LIN {X 0,Y 451.466,Z 366.784,A -85,B 0,C 180,E1 -8791.654,E2 -8791.654} C_VEL
LIN {X 0,Y 453.268,Z 375.362,A -85,B 0,C 180,E1 -8793.527,E2 -8793.527} C_VEL
LIN {X 0,Y 451.61,Z 393.058,A -85,B 0,C 180,E1 -8796.66,E2 -8796.66} C_VEL
LIN {X 0,Y 451.152,Z 398.451,A -85,B 0,C 180,E1 -8797.534,E2 -8797.534} C_VEL
LIN {X 0,Y 454.645,Z 414.595,A -85,B 0,C 180,E1 -8798.223,E2 -8798.223} C_VEL
LIN {X 0,Y 455.627,Z 420.756,A -85,B 0,C 180,E1 -8798.444,E2 -8798.444} C_VEL
LIN {X 0,Y 452.915,Z 505.565,A -85,B 0,C 180,E1 -8800.275,E2 -8800.275} C_VEL
LIN {X 0,Y 452.018,Z 542.086,A -85,B 0,C 180,E1 -8801.061,E2 -8801.061} C_VEL
LIN {X 0,Y 451.407,Z 557.431,A -85,B 0,C 180,E1 -8801.582,E2 -8801.582} C_VEL
LIN {X 0,Y 450.85,Z 571.274,A -85,B 0,C 180,E1 -8802.243,E2 -8802.243} C_VEL
LIN {X 0,Y 450.077,Z 585.059,A -85,B 0,C 180,E1 -8803.092,E2 -8803.092} C_VEL
LIN {X 0,Y 449.288,Z 598.112,A -85,B 0,C 180,E1 -8804.113,E2 -8804.113} C_VEL
LIN {X 0,Y 448.6,Z 609.92,A -85,B 0,C 180,E1 -8805.251,E2 -8805.251} C_VEL
LIN {X 0,Y 447.822,Z 620.998,A -85,B 0,C 180,E1 -8806.544,E2 -8806.544} C_VEL
LIN {X 0,Y 447.203,Z 631.086,A -85,B 0,C 180,E1 -8807.981,E2 -8807.981} C_VEL
LIN {X 0,Y 446.693,Z 638.983,A -85,B 0,C 180,E1 -8809.347,E2 -8809.347} C_VEL
LIN {X 0,Y 446.266,Z 646.534,A -85,B 0,C 180,E1 -8810.939,E2 -8810.939} C_VEL
LIN {X 0,Y 445.957,Z 651.754,A -85,B 0,C 180,E1 -8812.302,E2 -8812.302} C_VEL
LIN {X 0,Y 445.838,Z 655.972,A -85,B 0,C 180,E1 -8813.665,E2 -8813.665} C_VEL
LIN {X 0,Y 445.563,Z 660.212,A -85,B 0,C 180,E1 -8815.477,E2 -8815.477} C_VEL
LIN {X 0,Y 445.511,Z 662.951,A -85,B 0,C 180,E1 -8817.288,E2 -8817.288} C_VEL
LIN {X 0,Y 445.425,Z 664.278,A -85,B 0,C 180,E1 -8819.096,E2 -8819.096} C_VEL
LIN {X 0,Y 445.408,Z 664.199,A -85,B 0,C 180,E1 -8820.904,E2 -8820.904} C_VEL
LIN {X 0,Y 445.492,Z 662.715,A -85,B 0,C 180,E1 -8822.713,E2 -8822.713} C_VEL
LIN {X 0,Y 445.553,Z 661.444,A -85,B 0,C 180,E1 -8823.618,E2 -8823.618} C_VEL
LIN {X 0,Y 445.637,Z 657.807,A -85,B 0,C 180,E1 -8825.43,E2 -8825.43} C_VEL
LIN {X 0,Y 445.752,Z 654.529,A -85,B 0,C 180,E1 -8826.647,E2 -8826.647} C_VEL
LIN {X 0,Y 445.941,Z 649.406,A -85,B 0,C 180,E1 -8828.154,E2 -8828.154} C_VEL
LIN {X 0,Y 446.291,Z 642.628,A -85,B 0,C 180,E1 -8829.746,E2 -8829.746} C_VEL
LIN {X 0,Y 446.76,Z 634.19,A -85,B 0,C 180,E1 -8831.341,E2 -8831.341} C_VEL
LIN {X 0,Y 447.284,Z 625.36,A -85,B 0,C 180,E1 -8832.708,E2 -8832.708} C_VEL
LIN {X 0,Y 447.905,Z 614.653,A -85,B 0,C 180,E1 -8834.076,E2 -8834.076} C_VEL
LIN {X 0,Y 448.625,Z 602.694,A -85,B 0,C 180,E1 -8835.329,E2 -8835.329} C_VEL
LIN {X 0,Y 449.347,Z 590.755,A -85,B 0,C 180,E1 -8836.352,E2 -8836.352} C_VEL
LIN {X 0,Y 450.048,Z 577.658,A -85,B 0,C 180,E1 -8837.26,E2 -8837.26} C_VEL
LIN {X 0,Y 450.686,Z 563.753,A -85,B 0,C 180,E1 -8838.012,E2 -8838.012} C_VEL
LIN {X 0,Y 451.198,Z 549.271,A -85,B 0,C 180,E1 -8838.592,E2 -8838.592} C_VEL
LIN {X 0,Y 451.622,Z 534.731,A -85,B 0,C 180,E1 -8838.986,E2 -8838.986} C_VEL
LIN {X 0,Y 453.696,Z 419.17,A -85,B 0,C 180,E1 -8841.144,E2 -8841.144} C_VEL
LIN {X 0,Y 449.714,Z 397.572,A -85,B 0,C 180,E1 -8841.791,E2 -8841.791} C_VEL
LIN {X 0,Y 450.922,Z 378.264,A -85,B 0,C 180,E1 -8844.886,E2 -8844.886} C_VEL
LIN {X 0,Y 451.344,Z 370.862,A -85,B 0,C 180,E1 -8846.097,E2 -8846.097} C_VEL
LIN {X 0,Y 448.252,Z 357.222,A -85,B 0,C 180,E1 -8848.597,E2 -8848.597} C_VEL
LIN {X 0,Y 446.449,Z 349.788,A -85,B 0,C 180,E1 -8850.024,E2 -8850.024} C_VEL
LIN {X 0,Y 446.416,Z 349.503,A -85,B 0,C 180,E1 -8850.251,E2 -8850.251} C_VEL
LIN {X 0,Y 446.425,Z 349.502,A -85,B 0,C 180,E1 -8853.449,E2 -8853.449} C_VEL
LIN {X 0,Y 446.391,Z 349.505,A -85,B 0,C 180,E1 -8856.747,E2 -8856.747} C_VEL
LIN {X 0,Y 446.392,Z 349.508,A -85,B 0,C 180,E1 -8860.204,E2 -8860.204} C_VEL
LIN {X 0,Y 446.38,Z 349.497,A -85,B 0,C 180,E1 -8863.594,E2 -8863.594} C_VEL
LIN {X 0,Y 446.378,Z 349.497,A -85,B 0,C 180,E1 -8866.406,E2 -8866.406} C_VEL
LIN {X 0,Y 446.387,Z 349.503,A -85,B 0,C 180,E1 -8869.796,E2 -8869.796} C_VEL
LIN {X 0,Y 446.391,Z 349.499,A -85,B 0,C 180,E1 -8873.253,E2 -8873.253} C_VEL
LIN {X 0,Y 446.425,Z 349.504,A -85,B 0,C 180,E1 -8876.551,E2 -8876.551} C_VEL
LIN {X 0,Y 446.449,Z 349.719,A -85,B 0,C 180,E1 -8877.761,E2 -8877.761} C_VEL
LIN {X 0,Y 450.776,Z 366.42,A -85,B 0,C 180,E1 -8880.498,E2 -8880.498} C_VEL
LIN {X 0,Y 452.483,Z 374.302,A -85,B 0,C 180,E1 -8881.723,E2 -8881.723} C_VEL
LIN {X 0,Y 451.989,Z 384.049,A -85,B 0,C 180,E1 -8883.058,E2 -8883.058} C_VEL
LIN {X 0,Y 451.215,Z 387.102,A -85,B 0,C 180,E1 -8883.428,E2 -8883.428} C_VEL
LIN {X 0,Y 448.155,Z 392.329,A -85,B 0,C 180,E1 -8883.945,E2 -8883.945} C_VEL
LIN {X 0,Y 445.622,Z 397.396,A -85,B 0,C 180,E1 -8884.337,E2 -8884.337} C_VEL
LIN {X 0,Y 445.361,Z 400.297,A -85,B 0,C 180,E1 -8884.478,E2 -8884.478} C_VEL
LIN {X 0,Y 445.453,Z 400.893,A -85,B 0,C 180,E1 -8884.498,E2 -8884.498} C_VEL
LIN {X 0,Y 449.746,Z 423.038,A -85,B 0,C 180,E1 -8885.141,E2 -8885.141} C_VEL
LIN {X 0,Y 449.819,Z 431.74,A -85,B 0,C 180,E1 -8885.295,E2 -8885.295} C_VEL
LIN {X 0,Y 447.9,Z 564.075,A -85,B 0,C 180,E1 -8887.483,E2 -8887.483} C_VEL
LIN {X 0,Y 447.321,Z 579.57,A -85,B 0,C 180,E1 -8887.902,E2 -8887.902} C_VEL
LIN {X 0,Y 446.707,Z 592.8,A -85,B 0,C 180,E1 -8888.419,E2 -8888.419} C_VEL
LIN {X 0,Y 445.871,Z 606.369,A -85,B 0,C 180,E1 -8889.107,E2 -8889.107} C_VEL
LIN {X 0,Y 444.82,Z 620.534,A -85,B 0,C 180,E1 -8890.021,E2 -8890.021} C_VEL
LIN {X 0,Y 443.782,Z 633.454,A -85,B 0,C 180,E1 -8891.055,E2 -8891.055} C_VEL
LIN {X 0,Y 442.744,Z 645.813,A -85,B 0,C 180,E1 -8892.256,E2 -8892.256} C_VEL
LIN {X 0,Y 441.736,Z 657.318,A -85,B 0,C 180,E1 -8893.596,E2 -8893.596} C_VEL
LIN {X 0,Y 440.866,Z 667.346,A -85,B 0,C 180,E1 -8894.986,E2 -8894.986} C_VEL
LIN {X 0,Y 440.023,Z 677.147,A -85,B 0,C 180,E1 -8896.609,E2 -8896.609} C_VEL
LIN {X 0,Y 439.507,Z 685.285,A -85,B 0,C 180,E1 -8898.236,E2 -8898.236} C_VEL
LIN {X 0,Y 438.932,Z 692.025,A -85,B 0,C 180,E1 -8899.856,E2 -8899.856} C_VEL
LIN {X 0,Y 438.616,Z 698.269,A -85,B 0,C 180,E1 -8901.708,E2 -8901.708} C_VEL
LIN {X 0,Y 438.366,Z 703.48,A -85,B 0,C 180,E1 -8903.722,E2 -8903.722} C_VEL
LIN {X 0,Y 438.3,Z 706.652,A -85,B 0,C 180,E1 -8905.401,E2 -8905.401} C_VEL
LIN {X 0,Y 438.287,Z 708.995,A -85,B 0,C 180,E1 -8907.243,E2 -8907.243} C_VEL
LIN {X 0,Y 438.228,Z 710.186,A -85,B 0,C 180,E1 -8909.081,E2 -8909.081} C_VEL
LIN {X 0,Y 438.228,Z 710.202,A -85,B 0,C 180,E1 -8910.919,E2 -8910.919} C_VEL
LIN {X 0,Y 438.287,Z 709.07,A -85,B 0,C 180,E1 -8912.757,E2 -8912.757} C_VEL
LIN {X 0,Y 438.301,Z 706.79,A -85,B 0,C 180,E1 -8914.598,E2 -8914.598} C_VEL
LIN {X 0,Y 438.447,Z 703.314,A -85,B 0,C 180,E1 -8916.442,E2 -8916.442} C_VEL
LIN {X 0,Y 438.612,Z 698.552,A -85,B 0,C 180,E1 -8918.291,E2 -8918.291} C_VEL
LIN {X 0,Y 438.909,Z 692.375,A -85,B 0,C 180,E1 -8920.145,E2 -8920.145} C_VEL
LIN {X 0,Y 439.513,Z 684.613,A -85,B 0,C 180,E1 -8921.998,E2 -8921.998} C_VEL
LIN {X 0,Y 440.083,Z 676.342,A -85,B 0,C 180,E1 -8923.624,E2 -8923.624} C_VEL
LIN {X 0,Y 440.95,Z 666.376,A -85,B 0,C 180,E1 -8925.247,E2 -8925.247} C_VEL
LIN {X 0,Y 441.854,Z 656.204,A -85,B 0,C 180,E1 -8926.637,E2 -8926.637} C_VEL
LIN {X 0,Y 442.904,Z 644.034,A -85,B 0,C 180,E1 -8928.024,E2 -8928.024} C_VEL
LIN {X 0,Y 443.966,Z 631.862,A -85,B 0,C 180,E1 -8929.176,E2 -8929.176} C_VEL
LIN {X 0,Y 444.99,Z 618.593,A -85,B 0,C 180,E1 -8930.211,E2 -8930.211} C_VEL
LIN {X 0,Y 445.971,Z 604.954,A -85,B 0,C 180,E1 -8931.069,E2 -8931.069} C_VEL
LIN {X 0,Y 446.807,Z 589.736,A -85,B 0,C 180,E1 -8931.815,E2 -8931.815} C_VEL
LIN {X 0,Y 447.52,Z 575.51,A -85,B 0,C 180,E1 -8932.324,E2 -8932.324} C_VEL
LIN {X 0,Y 447.954,Z 560.083,A -85,B 0,C 180,E1 -8932.697,E2 -8932.697} C_VEL
LIN {X 0,Y 449.98,Z 425.271,A -85,B 0,C 180,E1 -8934.901,E2 -8934.901} C_VEL
LIN {X 0,Y 448.818,Z 417.732,A -85,B 0,C 180,E1 -8935.1,E2 -8935.1} C_VEL
LIN {X 0,Y 444.78,Z 397.136,A -85,B 0,C 180,E1 -8935.727,E2 -8935.727} C_VEL
LIN {X 0,Y 445.685,Z 378.356,A -85,B 0,C 180,E1 -8938.234,E2 -8938.234} C_VEL
LIN {X 0,Y 445.495,Z 374.677,A -85,B 0,C 180,E1 -8938.761,E2 -8938.761} C_VEL
LIN {X 0,Y 441.858,Z 359.718,A -85,B 0,C 180,E1 -8941.184,E2 -8941.184} C_VEL
LIN {X 0,Y 439.398,Z 350.524,A -85,B 0,C 180,E1 -8942.744,E2 -8942.744} C_VEL
LIN {X 0,Y 439.363,Z 350.373,A -85,B 0,C 180,E1 -8946.288,E2 -8946.288} C_VEL
LIN {X 0,Y 439.348,Z 350.379,A -85,B 0,C 180,E1 -8948.599,E2 -8948.599} C_VEL
LIN {X 0,Y 439.345,Z 350.381,A -85,B 0,C 180,E1 -8952.21,E2 -8952.21} C_VEL
LIN {X 0,Y 439.375,Z 350.376,A -85,B 0,C 180,E1 -8955.267,E2 -8955.267} C_VEL
LIN {X 0,Y 439.362,Z 350.38,A -85,B 0,C 180,E1 -8958.747,E2 -8958.747} C_VEL
LIN {X 0,Y 439.356,Z 350.379,A -85,B 0,C 180,E1 -8961.611,E2 -8961.611} C_VEL
LIN {X 0,Y 439.393,Z 350.369,A -85,B 0,C 180,E1 -8964.843,E2 -8964.843} C_VEL
LIN {X 0,Y 439.369,Z 350.372,A -85,B 0,C 180,E1 -8968.139,E2 -8968.139} C_VEL
LIN {X 0,Y 439.404,Z 350.374,A -85,B 0,C 180,E1 -8971.605,E2 -8971.605} C_VEL
LIN {X 0,Y 439.366,Z 350.378,A -85,B 0,C 180,E1 -8974.413,E2 -8974.413} C_VEL
LIN {X 0,Y 439.363,Z 350.373,A -85,B 0,C 180,E1 -8977.424,E2 -8977.424} C_VEL
LIN {X 0,Y 439.441,Z 350.368,A -85,B 0,C 180,E1 -8980.663,E2 -8980.663} C_VEL
LIN {X 0,Y 439.463,Z 350.363,A -85,B 0,C 180,E1 -8984.224,E2 -8984.224} C_VEL
LIN {X 0,Y 439.484,Z 350.356,A -85,B 0,C 180,E1 -8988.001,E2 -8988.001} C_VEL
LIN {X 0,Y 439.504,Z 350.365,A -85,B 0,C 180,E1 -8991.725,E2 -8991.725} C_VEL
LIN {X 0,Y 439.619,Z 350.337,A -85,B 0,C 180,E1 -8994.496,E2 -8994.496} C_VEL
LIN {X 0,Y 439.631,Z 350.345,A -85,B 0,C 180,E1 -8998.168,E2 -8998.168} C_VEL
LIN {X 0,Y 439.761,Z 350.323,A -85,B 0,C 180,E1 -9000,E2 -9000} C_VEL
LIN {X 0,Y 439.634,Z 350.337,A -85,B 0,C 180,E1 -9002.749,E2 -9002.749} C_VEL
LIN {X 0,Y 439.593,Z 350.344,A -85,B 0,C 180,E1 -9006.425,E2 -9006.425} C_VEL
LIN {X 0,Y 439.497,Z 350.356,A -85,B 0,C 180,E1 -9009.202,E2 -9009.202} C_VEL
LIN {X 0,Y 439.466,Z 350.361,A -85,B 0,C 180,E1 -9012.938,E2 -9012.938} C_VEL
LIN {X 0,Y 439.447,Z 350.367,A -85,B 0,C 180,E1 -9016.348,E2 -9016.348} C_VEL
LIN {X 0,Y 439.402,Z 350.365,A -85,B 0,C 180,E1 -9019.626,E2 -9019.626} C_VEL
LIN {X 0,Y 439.365,Z 350.379,A -85,B 0,C 180,E1 -9022.575,E2 -9022.575} C_VEL
LIN {X 0,Y 439.4,Z 350.371,A -85,B 0,C 180,E1 -9025.585,E2 -9025.585} C_VEL
LIN {X 0,Y 439.418,Z 350.374,A -85,B 0,C 180,E1 -9028.673,E2 -9028.673} C_VEL
LIN {X 0,Y 439.37,Z 350.378,A -85,B 0,C 180,E1 -9032.03,E2 -9032.03} C_VEL
LIN {X 0,Y 439.394,Z 350.376,A -85,B 0,C 180,E1 -9035.34,E2 -9035.34} C_VEL
LIN {X 0,Y 439.375,Z 350.366,A -85,B 0,C 180,E1 -9038.596,E2 -9038.596} C_VEL
LIN {X 0,Y 439.388,Z 350.355,A -85,B 0,C 180,E1 -9041.257,E2 -9041.257} C_VEL
LIN {X 0,Y 439.405,Z 350.373,A -85,B 0,C 180,E1 -9044.729,E2 -9044.729} C_VEL
LIN {X 0,Y 439.395,Z 350.364,A -85,B 0,C 180,E1 -9047.796,E2 -9047.796} C_VEL
LIN {X 0,Y 439.43,Z 350.372,A -85,B 0,C 180,E1 -9050.228,E2 -9050.228} C_VEL
LIN {X 0,Y 439.373,Z 350.378,A -85,B 0,C 180,E1 -9053.713,E2 -9053.713} C_VEL
LIN {X 0,Y 439.384,Z 350.38,A -85,B 0,C 180,E1 -9057.055,E2 -9057.055} C_VEL
LIN {X 0,Y 439.441,Z 350.626,A -85,B 0,C 180,E1 -9057.582,E2 -9057.582} C_VEL
LIN {X 0,Y 444.398,Z 368.974,A -85,B 0,C 180,E1 -9060.643,E2 -9060.643} C_VEL
LIN {X 0,Y 446.318,Z 376.633,A -85,B 0,C 180,E1 -9061.861,E2 -9061.861} C_VEL
LIN {X 0,Y 445.263,Z 391.914,A -85,B 0,C 180,E1 -9063.961,E2 -9063.961} C_VEL
LIN {X 0,Y 444.918,Z 396.826,A -85,B 0,C 180,E1 -9064.6,E2 -9064.6} C_VEL
LIN {X 0,Y 449.267,Z 422.728,A -85,B 0,C 180,E1 -9065.326,E2 -9065.326} C_VEL
LIN {X 0,Y 447.201,Z 564.707,A -85,B 0,C 180,E1 -9067.659,E2 -9067.659} C_VEL
LIN {X 0,Y 446.7,Z 580.228,A -85,B 0,C 180,E1 -9068.093,E2 -9068.093} C_VEL
LIN {X 0,Y 446.002,Z 594.377,A -85,B 0,C 180,E1 -9068.664,E2 -9068.664} C_VEL
LIN {X 0,Y 445.107,Z 608.773,A -85,B 0,C 180,E1 -9069.432,E2 -9069.432} C_VEL
LIN {X 0,Y 444.194,Z 622.326,A -85,B 0,C 180,E1 -9070.354,E2 -9070.354} C_VEL
LIN {X 0,Y 443.208,Z 634.778,A -85,B 0,C 180,E1 -9071.39,E2 -9071.39} C_VEL
LIN {X 0,Y 442.171,Z 647.145,A -85,B 0,C 180,E1 -9072.635,E2 -9072.635} C_VEL
LIN {X 0,Y 441.225,Z 658.798,A -85,B 0,C 180,E1 -9074.052,E2 -9074.052} C_VEL
LIN {X 0,Y 440.412,Z 668.389,A -85,B 0,C 180,E1 -9075.444,E2 -9075.444} C_VEL
LIN {X 0,Y 439.683,Z 677.782,A -85,B 0,C 180,E1 -9077.069,E2 -9077.069} C_VEL
LIN {X 0,Y 439.216,Z 685.58,A -85,B 0,C 180,E1 -9078.696,E2 -9078.696} C_VEL
LIN {X 0,Y 438.785,Z 692.041,A -85,B 0,C 180,E1 -9080.318,E2 -9080.318} C_VEL
LIN {X 0,Y 438.531,Z 697.96,A -85,B 0,C 180,E1 -9082.171,E2 -9082.171} C_VEL
LIN {X 0,Y 438.372,Z 701.809,A -85,B 0,C 180,E1 -9083.712,E2 -9083.712} C_VEL
LIN {X 0,Y 438.3,Z 704.995,A -85,B 0,C 180,E1 -9085.402,E2 -9085.402} C_VEL
LIN {X 0,Y 438.341,Z 707.327,A -85,B 0,C 180,E1 -9087.243,E2 -9087.243} C_VEL
LIN {X 0,Y 438.229,Z 708.501,A -85,B 0,C 180,E1 -9089.081,E2 -9089.081} C_VEL
LIN {X 0,Y 438.23,Z 708.501,A -85,B 0,C 180,E1 -9090.919,E2 -9090.919} C_VEL
LIN {X 0,Y 438.346,Z 707.329,A -85,B 0,C 180,E1 -9092.757,E2 -9092.757} C_VEL
LIN {X 0,Y 438.3,Z 704.996,A -85,B 0,C 180,E1 -9094.599,E2 -9094.599} C_VEL
LIN {X 0,Y 438.367,Z 701.445,A -85,B 0,C 180,E1 -9096.444,E2 -9096.444} C_VEL
LIN {X 0,Y 438.593,Z 696.593,A -85,B 0,C 180,E1 -9098.292,E2 -9098.292} C_VEL
LIN {X 0,Y 438.853,Z 690.314,A -85,B 0,C 180,E1 -9100.146,E2 -9100.146} C_VEL
LIN {X 0,Y 439.353,Z 683.524,A -85,B 0,C 180,E1 -9101.768,E2 -9101.768} C_VEL
LIN {X 0,Y 439.925,Z 675.307,A -85,B 0,C 180,E1 -9103.394,E2 -9103.394} C_VEL
LIN {X 0,Y 440.68,Z 665.392,A -85,B 0,C 180,E1 -9105.02,E2 -9105.02} C_VEL
LIN {X 0,Y 441.488,Z 655.224,A -85,B 0,C 180,E1 -9106.413,E2 -9106.413} C_VEL
LIN {X 0,Y 442.536,Z 643.3,A -85,B 0,C 180,E1 -9107.777,E2 -9107.777} C_VEL
LIN {X 0,Y 443.506,Z 630.878,A -85,B 0,C 180,E1 -9108.957,E2 -9108.957} C_VEL
LIN {X 0,Y 444.53,Z 617.563,A -85,B 0,C 180,E1 -9109.992,E2 -9109.992} C_VEL
LIN {X 0,Y 445.576,Z 602.772,A -85,B 0,C 180,E1 -9110.908,E2 -9110.908} C_VEL
LIN {X 0,Y 446.337,Z 588.561,A -85,B 0,C 180,E1 -9111.588,E2 -9111.588} C_VEL
LIN {X 0,Y 446.987,Z 573.017,A -85,B 0,C 180,E1 -9112.129,E2 -9112.129} C_VEL
LIN {X 0,Y 447.396,Z 556.928,A -85,B 0,C 180,E1 -9112.483,E2 -9112.483} C_VEL
LIN {X 0,Y 448.953,Z 450.43,A -85,B 0,C 180,E1 -9114.24,E2 -9114.24} C_VEL
LIN {X 0,Y 449.701,Z 421.272,A -85,B 0,C 180,E1 -9114.867,E2 -9114.867} C_VEL
LIN {X 0,Y 446.922,Z 403.458,A -85,B 0,C 180,E1 -9115.502,E2 -9115.502} C_VEL
LIN {X 0,Y 445.941,Z 398.268,A -85,B 0,C 180,E1 -9115.743,E2 -9115.743} C_VEL
LIN {X 0,Y 447.865,Z 381.434,A -85,B 0,C 180,E1 -9118.25,E2 -9118.25} C_VEL
LIN {X 0,Y 447.719,Z 378.874,A -85,B 0,C 180,E1 -9118.688,E2 -9118.688} C_VEL
LIN {X 0,Y 445.308,Z 368.642,A -85,B 0,C 180,E1 -9120.742,E2 -9120.742} C_VEL
LIN {X 0,Y 442.439,Z 359.291,A -85,B 0,C 180,E1 -9122.926,E2 -9122.926} C_VEL
LIN {X 0,Y 439.958,Z 352.426,A -85,B 0,C 180,E1 -9124.825,E2 -9124.825} C_VEL
LIN {X 0,Y 439.383,Z 350.43,A -85,B 0,C 180,E1 -9125.514,E2 -9125.514} C_VEL
LIN {X 0,Y 439.384,Z 350.381,A -85,B 0,C 180,E1 -9128.595,E2 -9128.595} C_VEL
LIN {X 0,Y 439.389,Z 350.38,A -85,B 0,C 180,E1 -9131.257,E2 -9131.257} C_VEL
LIN {X 0,Y 439.399,Z 350.379,A -85,B 0,C 180,E1 -9134.73,E2 -9134.73} C_VEL
LIN {X 0,Y 439.385,Z 350.38,A -85,B 0,C 180,E1 -9137.794,E2 -9137.794} C_VEL
LIN {X 0,Y 439.389,Z 350.38,A -85,B 0,C 180,E1 -9140.223,E2 -9140.223} C_VEL
LIN {X 0,Y 439.372,Z 350.382,A -85,B 0,C 180,E1 -9143.713,E2 -9143.713} C_VEL
LIN {X 0,Y 439.416,Z 350.546,A -85,B 0,C 180,E1 -9146.21,E2 -9146.21} C_VEL
LIN {X 0,Y 441.608,Z 357.326,A -85,B 0,C 180,E1 -9148.32,E2 -9148.32} C_VEL
LIN {X 0,Y 444.133,Z 365.947,A -85,B 0,C 180,E1 -9150.624,E2 -9150.624} C_VEL
LIN {X 0,Y 446.299,Z 375.378,A -85,B 0,C 180,E1 -9152.828,E2 -9152.828} C_VEL
LIN {X 0,Y 446.724,Z 377.823,A -85,B 0,C 180,E1 -9153.361,E2 -9153.361} C_VEL
LIN {X 0,Y 444.905,Z 395.726,A -85,B 0,C 180,E1 -9156.583,E2 -9156.583} C_VEL
LIN {X 0,Y 444.666,Z 398.418,A -85,B 0,C 180,E1 -9157.023,E2 -9157.023} C_VEL
LIN {X 0,Y 448.187,Z 414.555,A -85,B 0,C 180,E1 -9157.754,E2 -9157.754} C_VEL
LIN {X 0,Y 449.331,Z 422.382,A -85,B 0,C 180,E1 -9158.045,E2 -9158.045} C_VEL
LIN {X 0,Y 446.474,Z 504.686,A -85,B 0,C 180,E1 -9159.889,E2 -9159.889} C_VEL
LIN {X 0,Y 445.46,Z 542.04,A -85,B 0,C 180,E1 -9160.717,E2 -9160.717} C_VEL
LIN {X 0,Y 444.789,Z 557.63,A -85,B 0,C 180,E1 -9161.256,E2 -9161.256} C_VEL
LIN {X 0,Y 444.144,Z 572.359,A -85,B 0,C 180,E1 -9161.976,E2 -9161.976} C_VEL
LIN {X 0,Y 443.324,Z 585.762,A -85,B 0,C 180,E1 -9162.827,E2 -9162.827} C_VEL
LIN {X 0,Y 442.486,Z 598.72,A -85,B 0,C 180,E1 -9163.862,E2 -9163.862} C_VEL
LIN {X 0,Y 441.767,Z 610.473,A -85,B 0,C 180,E1 -9165.018,E2 -9165.018} C_VEL
LIN {X 0,Y 440.936,Z 621.682,A -85,B 0,C 180,E1 -9166.353,E2 -9166.353} C_VEL
LIN {X 0,Y 440.26,Z 631.568,A -85,B 0,C 180,E1 -9167.789,E2 -9167.789} C_VEL
LIN {X 0,Y 439.714,Z 639.451,A -85,B 0,C 180,E1 -9169.176,E2 -9169.176} C_VEL
LIN {X 0,Y 439.268,Z 646.975,A -85,B 0,C 180,E1 -9170.794,E2 -9170.794} C_VEL
LIN {X 0,Y 438.937,Z 652.19,A -85,B 0,C 180,E1 -9172.178,E2 -9172.178} C_VEL
LIN {X 0,Y 438.726,Z 657.628,A -85,B 0,C 180,E1 -9174.023,E2 -9174.023} C_VEL
LIN {X 0,Y 438.487,Z 660.621,A -85,B 0,C 180,E1 -9175.404,E2 -9175.404} C_VEL
LIN {X 0,Y 438.52,Z 662.157,A -85,B 0,C 180,E1 -9176.325,E2 -9176.325} C_VEL
LIN {X 0,Y 438.384,Z 664.168,A -85,B 0,C 180,E1 -9178.163,E2 -9178.163} C_VEL
LIN {X 0,Y 438.321,Z 664.766,A -85,B 0,C 180,E1 -9180,E2 -9180} C_VEL
LIN {X 0,Y 438.356,Z 663.945,A -85,B 0,C 180,E1 -9181.838,E2 -9181.838} C_VEL
LIN {X 0,Y 438.458,Z 661.718,A -85,B 0,C 180,E1 -9183.676,E2 -9183.676} C_VEL
LIN {X 0,Y 438.587,Z 658.035,A -85,B 0,C 180,E1 -9185.517,E2 -9185.517} C_VEL
LIN {X 0,Y 438.705,Z 654.282,A -85,B 0,C 180,E1 -9186.9,E2 -9186.9} C_VEL
LIN {X 0,Y 438.89,Z 649.55,A -85,B 0,C 180,E1 -9188.286,E2 -9188.286} C_VEL
LIN {X 0,Y 439.259,Z 642.708,A -85,B 0,C 180,E1 -9189.904,E2 -9189.904} C_VEL
LIN {X 0,Y 439.785,Z 634.172,A -85,B 0,C 180,E1 -9191.523,E2 -9191.523} C_VEL
LIN {X 0,Y 440.291,Z 625.257,A -85,B 0,C 180,E1 -9192.913,E2 -9192.913} C_VEL
LIN {X 0,Y 440.969,Z 614.452,A -85,B 0,C 180,E1 -9194.302,E2 -9194.302} C_VEL
LIN {X 0,Y 441.731,Z 602.379,A -85,B 0,C 180,E1 -9195.574,E2 -9195.574} C_VEL
LIN {X 0,Y 442.498,Z 590.311,A -85,B 0,C 180,E1 -9196.612,E2 -9196.612} C_VEL
LIN {X 0,Y 443.209,Z 577.038,A -85,B 0,C 180,E1 -9197.535,E2 -9197.535} C_VEL
LIN {X 0,Y 443.855,Z 563.864,A -85,B 0,C 180,E1 -9198.25,E2 -9198.25} C_VEL
LIN {X 0,Y 444.362,Z 549.683,A -85,B 0,C 180,E1 -9198.829,E2 -9198.829} C_VEL
LIN {X 0,Y 444.815,Z 535.354,A -85,B 0,C 180,E1 -9199.228,E2 -9199.228} C_VEL
LIN {X 0,Y 447.005,Z 420.277,A -85,B 0,C 180,E1 -9201.436,E2 -9201.436} C_VEL
LIN {X 0,Y 442.912,Z 397.889,A -85,B 0,C 180,E1 -9202.107,E2 -9202.107} C_VEL
LIN {X 0,Y 443.97,Z 381.108,A -85,B 0,C 180,E1 -9204.803,E2 -9204.803} C_VEL
LIN {X 0,Y 444.552,Z 373.397,A -85,B 0,C 180,E1 -9206.071,E2 -9206.071} C_VEL
LIN {X 0,Y 443.162,Z 366.192,A -85,B 0,C 180,E1 -9207.381,E2 -9207.381} C_VEL
LIN {X 0,Y 439.438,Z 350.774,A -85,B 0,C 180,E1 -9210.321,E2 -9210.321} C_VEL
LIN {X 0,Y 439.36,Z 350.41,A -85,B 0,C 180,E1 -9210.481,E2 -9210.481} C_VEL
LIN {X 0,Y 439.354,Z 350.385,A -85,B 0,C 180,E1 -9214.047,E2 -9214.047} C_VEL
LIN {X 0,Y 439.336,Z 350.384,A -85,B 0,C 180,E1 -9216.885,E2 -9216.885} C_VEL
LIN {X 0,Y 439.346,Z 350.385,A -85,B 0,C 180,E1 -9219.84,E2 -9219.84} C_VEL
LIN {X 0,Y 439.328,Z 350.371,A -85,B 0,C 180,E1 -9222.619,E2 -9222.619} C_VEL
LIN {X 0,Y 439.373,Z 350.379,A -85,B 0,C 180,E1 -9225.267,E2 -9225.267} C_VEL
LIN {X 0,Y 439.358,Z 350.382,A -85,B 0,C 180,E1 -9228.748,E2 -9228.748} C_VEL
LIN {X 0,Y 439.352,Z 350.381,A -85,B 0,C 180,E1 -9231.612,E2 -9231.612} C_VEL
LIN {X 0,Y 439.387,Z 350.378,A -85,B 0,C 180,E1 -9234.843,E2 -9234.843} C_VEL
LIN {X 0,Y 439.375,Z 350.524,A -85,B 0,C 180,E1 -9237.348,E2 -9237.348} C_VEL
LIN {X 0,Y 443.672,Z 366.741,A -85,B 0,C 180,E1 -9240.068,E2 -9240.068} C_VEL
LIN {X 0,Y 445.716,Z 375.854,A -85,B 0,C 180,E1 -9241.512,E2 -9241.512} C_VEL
LIN {X 0,Y 444.864,Z 394.937,A -85,B 0,C 180,E1 -9244.094,E2 -9244.094} C_VEL
LIN {X 0,Y 444.806,Z 397.613,A -85,B 0,C 180,E1 -9244.394,E2 -9244.394} C_VEL
LIN {X 0,Y 445.453,Z 400.893,A -85,B 0,C 180,E1 -9244.498,E2 -9244.498} C_VEL
LIN {X 0,Y 446.038,Z 406.682,A -85,B 0,C 180,E1 -9244.635,E2 -9244.635} C_VEL
LIN {X 0,Y 445.258,Z 416.52,A -85,B 0,C 180,E1 -9244.76,E2 -9244.76} C_VEL
LIN {X 0,Y 444.062,Z 424.472,A -85,B 0,C 180,E1 -9244.827,E2 -9244.827} C_VEL
LIN {X 0,Y 443.363,Z 432.441,A -85,B 0,C 180,E1 -9244.925,E2 -9244.925} C_VEL
LIN {X 0,Y 441.356,Z 563.988,A -85,B 0,C 180,E1 -9247.13,E2 -9247.13} C_VEL
LIN {X 0,Y 440.766,Z 578.845,A -85,B 0,C 180,E1 -9247.532,E2 -9247.532} C_VEL
LIN {X 0,Y 440.076,Z 592.717,A -85,B 0,C 180,E1 -9248.075,E2 -9248.075} C_VEL
LIN {X 0,Y 439.218,Z 606.337,A -85,B 0,C 180,E1 -9248.775,E2 -9248.775} C_VEL
LIN {X 0,Y 438.139,Z 620.508,A -85,B 0,C 180,E1 -9249.703,E2 -9249.703} C_VEL
LIN {X 0,Y 437.043,Z 633.431,A -85,B 0,C 180,E1 -9250.752,E2 -9250.752} C_VEL
LIN {X 0,Y 435.866,Z 646.524,A -85,B 0,C 180,E1 -9252.051,E2 -9252.051} C_VEL
LIN {X 0,Y 434.865,Z 657.3,A -85,B 0,C 180,E1 -9253.33,E2 -9253.33} C_VEL
LIN {X 0,Y 433.968,Z 667.329,A -85,B 0,C 180,E1 -9254.742,E2 -9254.742} C_VEL
LIN {X 0,Y 433.056,Z 677.131,A -85,B 0,C 180,E1 -9256.389,E2 -9256.389} C_VEL
LIN {X 0,Y 432.423,Z 686.315,A -85,B 0,C 180,E1 -9258.278,E2 -9258.278} C_VEL
LIN {X 0,Y 431.816,Z 693.728,A -85,B 0,C 180,E1 -9260.16,E2 -9260.16} C_VEL
LIN {X 0,Y 431.483,Z 699.612,A -85,B 0,C 180,E1 -9262.042,E2 -9262.042} C_VEL
LIN {X 0,Y 431.266,Z 703.781,A -85,B 0,C 180,E1 -9263.758,E2 -9263.758} C_VEL
LIN {X 0,Y 431.225,Z 706.638,A -85,B 0,C 180,E1 -9265.326,E2 -9265.326} C_VEL
LIN {X 0,Y 431.182,Z 708.981,A -85,B 0,C 180,E1 -9267.197,E2 -9267.197} C_VEL
LIN {X 0,Y 431.146,Z 710.173,A -85,B 0,C 180,E1 -9269.066,E2 -9269.066} C_VEL
LIN {X 0,Y 431.146,Z 710.188,A -85,B 0,C 180,E1 -9270.934,E2 -9270.934} C_VEL
LIN {X 0,Y 431.182,Z 709.055,A -85,B 0,C 180,E1 -9272.803,E2 -9272.803} C_VEL
LIN {X 0,Y 431.228,Z 706.776,A -85,B 0,C 180,E1 -9274.674,E2 -9274.674} C_VEL
LIN {X 0,Y 431.372,Z 703.299,A -85,B 0,C 180,E1 -9276.548,E2 -9276.548} C_VEL
LIN {X 0,Y 431.559,Z 698.535,A -85,B 0,C 180,E1 -9278.428,E2 -9278.428} C_VEL
LIN {X 0,Y 431.868,Z 692.357,A -85,B 0,C 180,E1 -9280.312,E2 -9280.312} C_VEL
LIN {X 0,Y 432.462,Z 685.691,A -85,B 0,C 180,E1 -9281.958,E2 -9281.958} C_VEL
LIN {X 0,Y 433.012,Z 677.615,A -85,B 0,C 180,E1 -9283.612,E2 -9283.612} C_VEL
LIN {X 0,Y 433.909,Z 667.916,A -85,B 0,C 180,E1 -9285.26,E2 -9285.26} C_VEL
LIN {X 0,Y 434.804,Z 657.98,A -85,B 0,C 180,E1 -9286.673,E2 -9286.673} C_VEL
LIN {X 0,Y 435.678,Z 648.071,A -85,B 0,C 180,E1 -9287.872,E2 -9287.872} C_VEL
LIN {X 0,Y 436.842,Z 635.672,A -85,B 0,C 180,E1 -9289.135,E2 -9289.135} C_VEL
LIN {X 0,Y 437.912,Z 623.225,A -85,B 0,C 180,E1 -9290.185,E2 -9290.185} C_VEL
LIN {X 0,Y 438.981,Z 609.727,A -85,B 0,C 180,E1 -9291.114,E2 -9291.114} C_VEL
LIN {X 0,Y 439.912,Z 595.638,A -85,B 0,C 180,E1 -9291.884,E2 -9291.884} C_VEL
LIN {X 0,Y 440.641,Z 581.153,A -85,B 0,C 180,E1 -9292.487,E2 -9292.487} C_VEL
LIN {X 0,Y 441.254,Z 566.778,A -85,B 0,C 180,E1 -9292.906,E2 -9292.906} C_VEL
LIN {X 0,Y 441.835,Z 533.359,A -85,B 0,C 180,E1 -9293.494,E2 -9293.494} C_VEL
LIN {X 0,Y 443.486,Z 424.86,A -85,B 0,C 180,E1 -9295.296,E2 -9295.296} C_VEL
LIN {X 0,Y 438.1,Z 397.116,A -85,B 0,C 180,E1 -9296.143,E2 -9296.143} C_VEL
LIN {X 0,Y 438.989,Z 379.693,A -85,B 0,C 180,E1 -9298.485,E2 -9298.485} C_VEL
LIN {X 0,Y 438.71,Z 376.309,A -85,B 0,C 180,E1 -9298.982,E2 -9298.982} C_VEL
LIN {X 0,Y 434.652,Z 359.737,A -85,B 0,C 180,E1 -9301.701,E2 -9301.701} C_VEL
LIN {X 0,Y 432.364,Z 351.363,A -85,B 0,C 180,E1 -9303.166,E2 -9303.166} C_VEL
LIN {X 0,Y 432.33,Z 351.249,A -85,B 0,C 180,E1 -9305.818,E2 -9305.818} C_VEL
LIN {X 0,Y 432.312,Z 351.253,A -85,B 0,C 180,E1 -9308.709,E2 -9308.709} C_VEL
LIN {X 0,Y 432.3,Z 351.263,A -85,B 0,C 180,E1 -9311.801,E2 -9311.801} C_VEL
LIN {X 0,Y 432.331,Z 351.255,A -85,B 0,C 180,E1 -9314.348,E2 -9314.348} C_VEL
LIN {X 0,Y 432.302,Z 351.261,A -85,B 0,C 180,E1 -9317.018,E2 -9317.018} C_VEL
LIN {X 0,Y 432.288,Z 351.264,A -85,B 0,C 180,E1 -9319.828,E2 -9319.828} C_VEL
LIN {X 0,Y 432.298,Z 351.26,A -85,B 0,C 180,E1 -9323.021,E2 -9323.021} C_VEL
LIN {X 0,Y 432.343,Z 351.257,A -85,B 0,C 180,E1 -9326,E2 -9326} C_VEL
LIN {X 0,Y 432.346,Z 351.25,A -85,B 0,C 180,E1 -9329.49,E2 -9329.49} C_VEL
LIN {X 0,Y 432.342,Z 351.249,A -85,B 0,C 180,E1 -9331.874,E2 -9331.874} C_VEL
LIN {X 0,Y 432.324,Z 351.255,A -85,B 0,C 180,E1 -9334.997,E2 -9334.997} C_VEL
LIN {X 0,Y 432.358,Z 351.244,A -85,B 0,C 180,E1 -9338.046,E2 -9338.046} C_VEL
LIN {X 0,Y 432.385,Z 351.249,A -85,B 0,C 180,E1 -9341.029,E2 -9341.029} C_VEL
LIN {X 0,Y 432.431,Z 351.237,A -85,B 0,C 180,E1 -9343.961,E2 -9343.961} C_VEL
LIN {X 0,Y 432.46,Z 351.232,A -85,B 0,C 180,E1 -9347.803,E2 -9347.803} C_VEL
LIN {X 0,Y 432.464,Z 351.243,A -85,B 0,C 180,E1 -9351.59,E2 -9351.59} C_VEL
LIN {X 0,Y 432.595,Z 351.212,A -85,B 0,C 180,E1 -9354.406,E2 -9354.406} C_VEL
LIN {X 0,Y 432.601,Z 351.221,A -85,B 0,C 180,E1 -9358.138,E2 -9358.138} C_VEL
LIN {X 0,Y 432.731,Z 351.199,A -85,B 0,C 180,E1 -9360,E2 -9360} C_VEL
LIN {X 0,Y 432.586,Z 351.215,A -85,B 0,C 180,E1 -9362.794,E2 -9362.794} C_VEL
LIN {X 0,Y 432.587,Z 351.222,A -85,B 0,C 180,E1 -9365.594,E2 -9365.594} C_VEL
LIN {X 0,Y 432.464,Z 351.226,A -85,B 0,C 180,E1 -9368.41,E2 -9368.41} C_VEL
LIN {X 0,Y 432.46,Z 351.233,A -85,B 0,C 180,E1 -9372.196,E2 -9372.196} C_VEL
LIN {X 0,Y 432.431,Z 351.241,A -85,B 0,C 180,E1 -9376.039,E2 -9376.039} C_VEL
LIN {X 0,Y 432.387,Z 351.238,A -85,B 0,C 180,E1 -9379.485,E2 -9379.485} C_VEL
LIN {X 0,Y 432.319,Z 351.261,A -85,B 0,C 180,E1 -9382.964,E2 -9382.964} C_VEL
LIN {X 0,Y 432.362,Z 351.247,A -85,B 0,C 180,E1 -9386.032,E2 -9386.032} C_VEL
LIN {X 0,Y 432.343,Z 351.249,A -85,B 0,C 180,E1 -9389.187,E2 -9389.187} C_VEL
LIN {X 0,Y 432.323,Z 351.257,A -85,B 0,C 180,E1 -9392.443,E2 -9392.443} C_VEL
LIN {X 0,Y 432.344,Z 351.255,A -85,B 0,C 180,E1 -9395.632,E2 -9395.632} C_VEL
LIN {X 0,Y 432.338,Z 351.239,A -85,B 0,C 180,E1 -9398.714,E2 -9398.714} C_VEL
LIN {X 0,Y 432.334,Z 351.243,A -85,B 0,C 180,E1 -9401.797,E2 -9401.797} C_VEL
LIN {X 0,Y 432.34,Z 351.255,A -85,B 0,C 180,E1 -9404.346,E2 -9404.346} C_VEL
LIN {X 0,Y 432.319,Z 351.236,A -85,B 0,C 180,E1 -9407.016,E2 -9407.016} C_VEL
LIN {X 0,Y 432.336,Z 351.255,A -85,B 0,C 180,E1 -9409.82,E2 -9409.82} C_VEL
LIN {X 0,Y 432.306,Z 351.262,A -85,B 0,C 180,E1 -9413.022,E2 -9413.022} C_VEL
LIN {X 0,Y 432.359,Z 351.256,A -85,B 0,C 180,E1 -9415.997,E2 -9415.997} C_VEL
LIN {X 0,Y 432.397,Z 351.504,A -85,B 0,C 180,E1 -9417.201,E2 -9417.201} C_VEL
LIN {X 0,Y 437.606,Z 370.765,A -85,B 0,C 180,E1 -9420.473,E2 -9420.473} C_VEL
LIN {X 0,Y 439.599,Z 379.254,A -85,B 0,C 180,E1 -9421.838,E2 -9421.838} C_VEL
LIN {X 0,Y 438.233,Z 396.054,A -85,B 0,C 180,E1 -9424.149,E2 -9424.149} C_VEL
LIN {X 0,Y 440.415,Z 408.746,A -85,B 0,C 180,E1 -9424.545,E2 -9424.545} C_VEL
LIN {X 0,Y 442.783,Z 424.102,A -85,B 0,C 180,E1 -9424.961,E2 -9424.961} C_VEL
LIN {X 0,Y 440.657,Z 564.835,A -85,B 0,C 180,E1 -9427.309,E2 -9427.309} C_VEL
LIN {X 0,Y 440.128,Z 580.292,A -85,B 0,C 180,E1 -9427.748,E2 -9427.748} C_VEL
LIN {X 0,Y 439.363,Z 594.732,A -85,B 0,C 180,E1 -9428.34,E2 -9428.34} C_VEL
LIN {X 0,Y 438.461,Z 608.817,A -85,B 0,C 180,E1 -9429.106,E2 -9429.106} C_VEL
LIN {X 0,Y 437.482,Z 622.362,A -85,B 0,C 180,E1 -9430.039,E2 -9430.039} C_VEL
LIN {X 0,Y 436.446,Z 634.808,A -85,B 0,C 180,E1 -9431.091,E2 -9431.091} C_VEL
LIN {X 0,Y 435.435,Z 646.391,A -85,B 0,C 180,E1 -9432.269,E2 -9432.269} C_VEL
LIN {X 0,Y 434.497,Z 657.047,A -85,B 0,C 180,E1 -9433.557,E2 -9433.557} C_VEL
LIN {X 0,Y 433.613,Z 666.931,A -85,B 0,C 180,E1 -9434.97,E2 -9434.97} C_VEL
LIN {X 0,Y 432.812,Z 676.575,A -85,B 0,C 180,E1 -9436.621,E2 -9436.621} C_VEL
LIN {X 0,Y 432.258,Z 684.593,A -85,B 0,C 180,E1 -9438.274,E2 -9438.274} C_VEL
LIN {X 0,Y 431.749,Z 692.058,A -85,B 0,C 180,E1 -9440.159,E2 -9440.159} C_VEL
LIN {X 0,Y 431.469,Z 697.976,A -85,B 0,C 180,E1 -9442.042,E2 -9442.042} C_VEL
LIN {X 0,Y 431.293,Z 702.081,A -85,B 0,C 180,E1 -9443.723,E2 -9443.723} C_VEL
LIN {X 0,Y 431.226,Z 705.009,A -85,B 0,C 180,E1 -9445.326,E2 -9445.326} C_VEL
LIN {X 0,Y 431.233,Z 707.341,A -85,B 0,C 180,E1 -9447.198,E2 -9447.198} C_VEL
LIN {X 0,Y 431.148,Z 708.514,A -85,B 0,C 180,E1 -9449.066,E2 -9449.066} C_VEL
LIN {X 0,Y 431.148,Z 708.515,A -85,B 0,C 180,E1 -9450.934,E2 -9450.934} C_VEL
LIN {X 0,Y 431.239,Z 707.343,A -85,B 0,C 180,E1 -9452.803,E2 -9452.803} C_VEL
LIN {X 0,Y 431.225,Z 705.01,A -85,B 0,C 180,E1 -9454.674,E2 -9454.674} C_VEL
LIN {X 0,Y 431.287,Z 701.459,A -85,B 0,C 180,E1 -9456.55,E2 -9456.55} C_VEL
LIN {X 0,Y 431.54,Z 696.608,A -85,B 0,C 180,E1 -9458.429,E2 -9458.429} C_VEL
LIN {X 0,Y 431.814,Z 690.329,A -85,B 0,C 180,E1 -9460.313,E2 -9460.313} C_VEL
LIN {X 0,Y 432.329,Z 683.54,A -85,B 0,C 180,E1 -9461.962,E2 -9461.962} C_VEL
LIN {X 0,Y 432.959,Z 675.323,A -85,B 0,C 180,E1 -9463.614,E2 -9463.614} C_VEL
LIN {X 0,Y 433.779,Z 665.411,A -85,B 0,C 180,E1 -9465.265,E2 -9465.265} C_VEL
LIN {X 0,Y 434.63,Z 655.244,A -85,B 0,C 180,E1 -9466.68,E2 -9466.68} C_VEL
LIN {X 0,Y 435.769,Z 643.102,A -85,B 0,C 180,E1 -9468.087,E2 -9468.087} C_VEL
LIN {X 0,Y 436.783,Z 630.903,A -85,B 0,C 180,E1 -9469.26,E2 -9469.26} C_VEL
LIN {X 0,Y 437.836,Z 617.593,A -85,B 0,C 180,E1 -9470.311,E2 -9470.311} C_VEL
LIN {X 0,Y 438.944,Z 602.809,A -85,B 0,C 180,E1 -9471.239,E2 -9471.239} C_VEL
LIN {X 0,Y 439.76,Z 588.31,A -85,B 0,C 180,E1 -9471.941,E2 -9471.941} C_VEL
LIN {X 0,Y 440.413,Z 573.165,A -85,B 0,C 180,E1 -9472.474,E2 -9472.474} C_VEL
LIN {X 0,Y 440.856,Z 557.05,A -85,B 0,C 180,E1 -9472.835,E2 -9472.835} C_VEL
LIN {X 0,Y 442.388,Z 459.964,A -85,B 0,C 180,E1 -9474.461,E2 -9474.461} C_VEL
LIN {X 0,Y 443.491,Z 422.194,A -85,B 0,C 180,E1 -9475.297,E2 -9475.297} C_VEL
LIN {X 0,Y 440.967,Z 405.481,A -85,B 0,C 180,E1 -9475.923,E2 -9475.923} C_VEL
LIN {X 0,Y 439.571,Z 398.326,A -85,B 0,C 180,E1 -9476.255,E2 -9476.255} C_VEL
LIN {X 0,Y 441.417,Z 383.429,A -85,B 0,C 180,E1 -9478.532,E2 -9478.532} C_VEL
LIN {X 0,Y 440.764,Z 379.01,A -85,B 0,C 180,E1 -9479.367,E2 -9479.367} C_VEL
LIN {X 0,Y 438.433,Z 369.61,A -85,B 0,C 180,E1 -9481.377,E2 -9481.377} C_VEL
LIN {X 0,Y 436.151,Z 362.168,A -85,B 0,C 180,E1 -9483.221,E2 -9483.221} C_VEL
LIN {X 0,Y 433.809,Z 355.65,A -85,B 0,C 180,E1 -9485.108,E2 -9485.108} C_VEL
LIN {X 0,Y 432.344,Z 351.339,A -85,B 0,C 180,E1 -9486.611,E2 -9486.611} C_VEL
LIN {X 0,Y 432.351,Z 351.257,A -85,B 0,C 180,E1 -9489.343,E2 -9489.343} C_VEL
LIN {X 0,Y 432.334,Z 351.258,A -85,B 0,C 180,E1 -9491.797,E2 -9491.797} C_VEL
LIN {X 0,Y 432.334,Z 351.259,A -85,B 0,C 180,E1 -9494.348,E2 -9494.348} C_VEL
LIN {X 0,Y 432.317,Z 351.261,A -85,B 0,C 180,E1 -9497.016,E2 -9497.016} C_VEL
LIN {X 0,Y 432.333,Z 351.259,A -85,B 0,C 180,E1 -9499.821,E2 -9499.821} C_VEL
LIN {X 0,Y 432.305,Z 351.263,A -85,B 0,C 180,E1 -9503.022,E2 -9503.022} C_VEL
LIN {X 0,Y 432.362,Z 351.414,A -85,B 0,C 180,E1 -9505.077,E2 -9505.077} C_VEL
LIN {X 0,Y 434.492,Z 357.608,A -85,B 0,C 180,E1 -9507.258,E2 -9507.258} C_VEL
LIN {X 0,Y 436.873,Z 365.418,A -85,B 0,C 180,E1 -9509.553,E2 -9509.553} C_VEL
LIN {X 0,Y 439.257,Z 375.188,A -85,B 0,C 180,E1 -9512.011,E2 -9512.011} C_VEL
LIN {X 0,Y 440.227,Z 380.402,A -85,B 0,C 180,E1 -9513.193,E2 -9513.193} C_VEL
LIN {X 0,Y 438.231,Z 398.139,A -85,B 0,C 180,E1 -9516.441,E2 -9516.441} C_VEL
LIN {X 0,Y 439.072,Z 402.188,A -85,B 0,C 180,E1 -9516.677,E2 -9516.677} C_VEL
LIN {X 0,Y 442.361,Z 417.597,A -85,B 0,C 180,E1 -9517.391,E2 -9517.391} C_VEL
LIN {X 0,Y 443.182,Z 422.812,A -85,B 0,C 180,E1 -9517.599,E2 -9517.599} C_VEL
LIN {X 0,Y 440.056,Z 504.347,A -85,B 0,C 180,E1 -9519.491,E2 -9519.491} C_VEL
LIN {X 0,Y 438.902,Z 543.015,A -85,B 0,C 180,E1 -9520.384,E2 -9520.384} C_VEL
LIN {X 0,Y 438.182,Z 558.408,A -85,B 0,C 180,E1 -9520.935,E2 -9520.935} C_VEL
LIN {X 0,Y 437.533,Z 572.066,A -85,B 0,C 180,E1 -9521.617,E2 -9521.617} C_VEL
LIN {X 0,Y 436.718,Z 585.008,A -85,B 0,C 180,E1 -9522.438,E2 -9522.438} C_VEL
LIN {X 0,Y 435.809,Z 598.141,A -85,B 0,C 180,E1 -9523.487,E2 -9523.487} C_VEL
LIN {X 0,Y 435.033,Z 610.031,A -85,B 0,C 180,E1 -9524.66,E2 -9524.66} C_VEL
LIN {X 0,Y 434.161,Z 620.844,A -85,B 0,C 180,E1 -9525.947,E2 -9525.947} C_VEL
LIN {X 0,Y 433.442,Z 630.611,A -85,B 0,C 180,E1 -9527.356,E2 -9527.356} C_VEL
LIN {X 0,Y 432.802,Z 638.716,A -85,B 0,C 180,E1 -9528.764,E2 -9528.764} C_VEL
LIN {X 0,Y 432.311,Z 646.463,A -85,B 0,C 180,E1 -9530.408,E2 -9530.408} C_VEL
LIN {X 0,Y 431.896,Z 652.66,A -85,B 0,C 180,E1 -9532.05,E2 -9532.05} C_VEL
LIN {X 0,Y 431.699,Z 656.844,A -85,B 0,C 180,E1 -9533.457,E2 -9533.457} C_VEL
LIN {X 0,Y 431.413,Z 661.045,A -85,B 0,C 180,E1 -9535.328,E2 -9535.328} C_VEL
LIN {X 0,Y 431.46,Z 662.569,A -85,B 0,C 180,E1 -9536.264,E2 -9536.264} C_VEL
LIN {X 0,Y 431.303,Z 664.557,A -85,B 0,C 180,E1 -9538.133,E2 -9538.133} C_VEL
LIN {X 0,Y 431.232,Z 665.116,A -85,B 0,C 180,E1 -9540,E2 -9540} C_VEL
LIN {X 0,Y 431.277,Z 664.254,A -85,B 0,C 180,E1 -9541.868,E2 -9541.868} C_VEL
LIN {X 0,Y 431.364,Z 661.984,A -85,B 0,C 180,E1 -9543.737,E2 -9543.737} C_VEL
LIN {X 0,Y 431.513,Z 658.25,A -85,B 0,C 180,E1 -9545.608,E2 -9545.608} C_VEL
LIN {X 0,Y 431.694,Z 652.957,A -85,B 0,C 180,E1 -9547.484,E2 -9547.484} C_VEL
LIN {X 0,Y 431.94,Z 647.829,A -85,B 0,C 180,E1 -9548.892,E2 -9548.892} C_VEL
LIN {X 0,Y 432.381,Z 640.454,A -85,B 0,C 180,E1 -9550.536,E2 -9550.536} C_VEL
LIN {X 0,Y 432.881,Z 632.73,A -85,B 0,C 180,E1 -9551.947,E2 -9551.947} C_VEL
LIN {X 0,Y 433.455,Z 623.269,A -85,B 0,C 180,E1 -9553.385,E2 -9553.385} C_VEL
LIN {X 0,Y 434.205,Z 612.214,A -85,B 0,C 180,E1 -9554.769,E2 -9554.769} C_VEL
LIN {X 0,Y 434.881,Z 600.809,A -85,B 0,C 180,E1 -9555.946,E2 -9555.946} C_VEL
LIN {X 0,Y 435.72,Z 588.265,A -85,B 0,C 180,E1 -9556.999,E2 -9556.999} C_VEL
LIN {X 0,Y 436.527,Z 574.516,A -85,B 0,C 180,E1 -9557.921,E2 -9557.921} C_VEL
LIN {X 0,Y 437.166,Z 559.956,A -85,B 0,C 180,E1 -9558.677,E2 -9558.677} C_VEL
LIN {X 0,Y 437.701,Z 545.674,A -85,B 0,C 180,E1 -9559.218,E2 -9559.218} C_VEL
LIN {X 0,Y 438.129,Z 530.368,A -85,B 0,C 180,E1 -9559.594,E2 -9559.594} C_VEL
LIN {X 0,Y 440.351,Z 421.289,A -85,B 0,C 180,E1 -9561.731,E2 -9561.731} C_VEL
LIN {X 0,Y 436.099,Z 397.76,A -85,B 0,C 180,E1 -9562.459,E2 -9562.459} C_VEL
LIN {X 0,Y 437.327,Z 379.438,A -85,B 0,C 180,E1 -9565.46,E2 -9565.46} C_VEL
LIN {X 0,Y 437.701,Z 374.813,A -85,B 0,C 180,E1 -9566.232,E2 -9566.232} C_VEL
LIN {X 0,Y 435.484,Z 364.439,A -85,B 0,C 180,E1 -9568.167,E2 -9568.167} C_VEL
LIN {X 0,Y 432.386,Z 351.714,A -85,B 0,C 180,E1 -9570.644,E2 -9570.644} C_VEL
LIN {X 0,Y 432.303,Z 351.266,A -85,B 0,C 180,E1 -9570.882,E2 -9570.882} C_VEL
LIN {X 0,Y 432.33,Z 351.26,A -85,B 0,C 180,E1 -9573.997,E2 -9573.997} C_VEL
LIN {X 0,Y 432.31,Z 351.259,A -85,B 0,C 180,E1 -9577.194,E2 -9577.194} C_VEL
LIN {X 0,Y 432.288,Z 351.265,A -85,B 0,C 180,E1 -9580.172,E2 -9580.172} C_VEL
LIN {X 0,Y 432.3,Z 351.247,A -85,B 0,C 180,E1 -9583.063,E2 -9583.063} C_VEL
LIN {X 0,Y 432.332,Z 351.257,A -85,B 0,C 180,E1 -9585.665,E2 -9585.665} C_VEL
LIN {X 0,Y 432.304,Z 351.263,A -85,B 0,C 180,E1 -9588.403,E2 -9588.403} C_VEL
LIN {X 0,Y 432.318,Z 351.26,A -85,B 0,C 180,E1 -9591.848,E2 -9591.848} C_VEL
LIN {X 0,Y 432.321,Z 351.255,A -85,B 0,C 180,E1 -9595.321,E2 -9595.321} C_VEL
LIN {X 0,Y 432.337,Z 351.476,A -85,B 0,C 180,E1 -9596.97,E2 -9596.97} C_VEL
LIN {X 0,Y 436.34,Z 366.42,A -85,B 0,C 180,E1 -9599.512,E2 -9599.512} C_VEL
LIN {X 0,Y 438.918,Z 377.432,A -85,B 0,C 180,E1 -9601.291,E2 -9601.291} C_VEL
LIN {X 0,Y 438.499,Z 388.448,A -85,B 0,C 180,E1 -9602.82,E2 -9602.82} C_VEL
LIN {X 0,Y 438.142,Z 397.417,A -85,B 0,C 180,E1 -9603.973,E2 -9603.973} C_VEL
LIN {X 0,Y 443.437,Z 424.846,A -85,B 0,C 180,E1 -9604.796,E2 -9604.796} C_VEL
LIN {X 0,Y 443.363,Z 432.441,A -85,B 0,C 180,E1 -9604.925,E2 -9604.925} C_VEL
LIN {X 0,Y 442.644,Z 438.297,A -85,B 0,C 180,E1 -9604.985,E2 -9604.985} C_VEL
LIN {X 0,Y 437.081,Z 457.362,A -85,B 0,C 180,E1 -9604.986,E2 -9604.986} C_VEL
LIN {X 0,Y 436.461,Z 463.211,A -85,B 0,C 180,E1 -9605.052,E2 -9605.052} C_VEL
LIN {X 0,Y 434.819,Z 563.902,A -85,B 0,C 180,E1 -9606.766,E2 -9606.766} C_VEL
LIN {X 0,Y 434.184,Z 579.373,A -85,B 0,C 180,E1 -9607.193,E2 -9607.193} C_VEL
LIN {X 0,Y 433.445,Z 593.531,A -85,B 0,C 180,E1 -9607.765,E2 -9607.765} C_VEL
LIN {X 0,Y 432.604,Z 606.305,A -85,B 0,C 180,E1 -9608.435,E2 -9608.435} C_VEL
LIN {X 0,Y 431.461,Z 620.481,A -85,B 0,C 180,E1 -9609.375,E2 -9609.375} C_VEL
LIN {X 0,Y 430.308,Z 633.408,A -85,B 0,C 180,E1 -9610.439,E2 -9610.439} C_VEL
LIN {X 0,Y 429.179,Z 645.56,A -85,B 0,C 180,E1 -9611.65,E2 -9611.65} C_VEL
LIN {X 0,Y 428.03,Z 657.282,A -85,B 0,C 180,E1 -9613.055,E2 -9613.055} C_VEL
LIN {X 0,Y 427.073,Z 667.312,A -85,B 0,C 180,E1 -9614.489,E2 -9614.489} C_VEL
LIN {X 0,Y 426.104,Z 677.115,A -85,B 0,C 180,E1 -9616.163,E2 -9616.163} C_VEL
LIN {X 0,Y 425.444,Z 685.255,A -85,B 0,C 180,E1 -9617.841,E2 -9617.841} C_VEL
LIN {X 0,Y 424.855,Z 691.996,A -85,B 0,C 180,E1 -9619.516,E2 -9619.516} C_VEL
LIN {X 0,Y 424.488,Z 698.241,A -85,B 0,C 180,E1 -9621.43,E2 -9621.43} C_VEL
LIN {X 0,Y 424.222,Z 703.076,A -85,B 0,C 180,E1 -9623.34,E2 -9623.34} C_VEL
LIN {X 0,Y 424.152,Z 706.625,A -85,B 0,C 180,E1 -9625.248,E2 -9625.248} C_VEL
LIN {X 0,Y 424.078,Z 708.968,A -85,B 0,C 180,E1 -9627.15,E2 -9627.15} C_VEL
LIN {X 0,Y 424.067,Z 710.159,A -85,B 0,C 180,E1 -9629.05,E2 -9629.05} C_VEL
LIN {X 0,Y 424.067,Z 710.174,A -85,B 0,C 180,E1 -9630.949,E2 -9630.949} C_VEL
LIN {X 0,Y 424.079,Z 709.041,A -85,B 0,C 180,E1 -9632.85,E2 -9632.85} C_VEL
LIN {X 0,Y 424.155,Z 706.761,A -85,B 0,C 180,E1 -9634.752,E2 -9634.752} C_VEL
LIN {X 0,Y 424.295,Z 703.283,A -85,B 0,C 180,E1 -9636.658,E2 -9636.658} C_VEL
LIN {X 0,Y 424.48,Z 698.518,A -85,B 0,C 180,E1 -9638.569,E2 -9638.569} C_VEL
LIN {X 0,Y 424.832,Z 692.339,A -85,B 0,C 180,E1 -9640.485,E2 -9640.485} C_VEL
LIN {X 0,Y 425.429,Z 685.672,A -85,B 0,C 180,E1 -9642.159,E2 -9642.159} C_VEL
LIN {X 0,Y 426.048,Z 677.595,A -85,B 0,C 180,E1 -9643.839,E2 -9643.839} C_VEL
LIN {X 0,Y 427.014,Z 667.893,A -85,B 0,C 180,E1 -9645.512,E2 -9645.512} C_VEL
LIN {X 0,Y 427.978,Z 657.955,A -85,B 0,C 180,E1 -9646.946,E2 -9646.946} C_VEL
LIN {X 0,Y 429.122,Z 646.159,A -85,B 0,C 180,E1 -9648.377,E2 -9648.377} C_VEL
LIN {X 0,Y 430.226,Z 634.377,A -85,B 0,C 180,E1 -9649.565,E2 -9649.565} C_VEL
LIN {X 0,Y 431.35,Z 621.647,A -85,B 0,C 180,E1 -9650.63,E2 -9650.63} C_VEL
LIN {X 0,Y 432.485,Z 607.763,A -85,B 0,C 180,E1 -9651.571,E2 -9651.571} C_VEL
LIN {X 0,Y 433.415,Z 593.738,A -85,B 0,C 180,E1 -9652.322,E2 -9652.322} C_VEL
LIN {X 0,Y 434.153,Z 579.668,A -85,B 0,C 180,E1 -9652.893,E2 -9652.893} C_VEL
LIN {X 0,Y 434.794,Z 563.942,A -85,B 0,C 180,E1 -9653.329,E2 -9653.329} C_VEL
LIN {X 0,Y 436.937,Z 435.773,A -85,B 0,C 180,E1 -9655.504,E2 -9655.504} C_VEL
LIN {X 0,Y 436.973,Z 425.414,A -85,B 0,C 180,E1 -9655.687,E2 -9655.687} C_VEL
LIN {X 0,Y 431.484,Z 397.43,A -85,B 0,C 180,E1 -9656.554,E2 -9656.554} C_VEL
LIN {X 0,Y 431.616,Z 392.802,A -85,B 0,C 180,E1 -9657.124,E2 -9657.124} C_VEL
LIN {X 0,Y 432.291,Z 380.675,A -85,B 0,C 180,E1 -9658.796,E2 -9658.796} C_VEL
LIN {X 0,Y 430.99,Z 373.972,A -85,B 0,C 180,E1 -9659.853,E2 -9659.853} C_VEL
LIN {X 0,Y 427.362,Z 359.675,A -85,B 0,C 180,E1 -9662.257,E2 -9662.257} C_VEL
LIN {X 0,Y 425.31,Z 352.269,A -85,B 0,C 180,E1 -9663.577,E2 -9663.577} C_VEL
LIN {X 0,Y 425.255,Z 352.131,A -85,B 0,C 180,E1 -9666.509,E2 -9666.509} C_VEL
LIN {X 0,Y 425.243,Z 352.129,A -85,B 0,C 180,E1 -9669.034,E2 -9669.034} C_VEL
LIN {X 0,Y 425.255,Z 352.135,A -85,B 0,C 180,E1 -9672.655,E2 -9672.655} C_VEL
LIN {X 0,Y 425.283,Z 352.131,A -85,B 0,C 180,E1 -9675.283,E2 -9675.283} C_VEL
LIN {X 0,Y 425.247,Z 352.139,A -85,B 0,C 180,E1 -9678.618,E2 -9678.618} C_VEL
LIN {X 0,Y 425.276,Z 352.13,A -85,B 0,C 180,E1 -9681.099,E2 -9681.099} C_VEL
LIN {X 0,Y 425.295,Z 352.125,A -85,B 0,C 180,E1 -9684.664,E2 -9684.664} C_VEL
LIN {X 0,Y 425.263,Z 352.129,A -85,B 0,C 180,E1 -9688.073,E2 -9688.073} C_VEL
LIN {X 0,Y 425.311,Z 352.133,A -85,B 0,C 180,E1 -9691.366,E2 -9691.366} C_VEL
LIN {X 0,Y 425.261,Z 352.135,A -85,B 0,C 180,E1 -9694.552,E2 -9694.552} C_VEL
LIN {X 0,Y 425.292,Z 352.124,A -85,B 0,C 180,E1 -9697.73,E2 -9697.73} C_VEL
LIN {X 0,Y 425.361,Z 352.122,A -85,B 0,C 180,E1 -9700.704,E2 -9700.704} C_VEL
LIN {X 0,Y 425.388,Z 352.111,A -85,B 0,C 180,E1 -9703.688,E2 -9703.688} C_VEL
LIN {X 0,Y 425.413,Z 352.112,A -85,B 0,C 180,E1 -9707.598,E2 -9707.598} C_VEL
LIN {X 0,Y 425.409,Z 352.119,A -85,B 0,C 180,E1 -9711.449,E2 -9711.449} C_VEL
LIN {X 0,Y 425.551,Z 352.089,A -85,B 0,C 180,E1 -9714.313,E2 -9714.313} C_VEL
LIN {X 0,Y 425.57,Z 352.097,A -85,B 0,C 180,E1 -9718.107,E2 -9718.107} C_VEL
LIN {X 0,Y 425.7,Z 352.074,A -85,B 0,C 180,E1 -9720,E2 -9720} C_VEL
LIN {X 0,Y 425.539,Z 352.093,A -85,B 0,C 180,E1 -9722.84,E2 -9722.84} C_VEL
LIN {X 0,Y 425.542,Z 352.098,A -85,B 0,C 180,E1 -9725.687,E2 -9725.687} C_VEL
LIN {X 0,Y 425.409,Z 352.104,A -85,B 0,C 180,E1 -9728.551,E2 -9728.551} C_VEL
LIN {X 0,Y 425.413,Z 352.111,A -85,B 0,C 180,E1 -9732.402,E2 -9732.402} C_VEL
LIN {X 0,Y 425.388,Z 352.118,A -85,B 0,C 180,E1 -9736.312,E2 -9736.312} C_VEL
LIN {X 0,Y 425.328,Z 352.117,A -85,B 0,C 180,E1 -9739.635,E2 -9739.635} C_VEL
LIN {X 0,Y 425.306,Z 352.129,A -85,B 0,C 180,E1 -9743.365,E2 -9743.365} C_VEL
LIN {X 0,Y 425.347,Z 352.125,A -85,B 0,C 180,E1 -9746.844,E2 -9746.844} C_VEL
LIN {X 0,Y 425.291,Z 352.123,A -85,B 0,C 180,E1 -9749.719,E2 -9749.719} C_VEL
LIN {X 0,Y 425.282,Z 352.135,A -85,B 0,C 180,E1 -9753.048,E2 -9753.048} C_VEL
LIN {X 0,Y 425.282,Z 352.133,A -85,B 0,C 180,E1 -9755.929,E2 -9755.929} C_VEL
LIN {X 0,Y 425.281,Z 352.11,A -85,B 0,C 180,E1 -9759.041,E2 -9759.041} C_VEL
LIN {X 0,Y 425.291,Z 352.123,A -85,B 0,C 180,E1 -9761.958,E2 -9761.958} C_VEL
LIN {X 0,Y 425.286,Z 352.122,A -85,B 0,C 180,E1 -9765.283,E2 -9765.283} C_VEL
LIN {X 0,Y 425.274,Z 352.13,A -85,B 0,C 180,E1 -9768.621,E2 -9768.621} C_VEL
LIN {X 0,Y 425.31,Z 352.135,A -85,B 0,C 180,E1 -9771.103,E2 -9771.103} C_VEL
LIN {X 0,Y 425.299,Z 352.135,A -85,B 0,C 180,E1 -9774.664,E2 -9774.664} C_VEL
LIN {X 0,Y 425.347,Z 352.363,A -85,B 0,C 180,E1 -9776.817,E2 -9776.817} C_VEL
LIN {X 0,Y 430.263,Z 370.521,A -85,B 0,C 180,E1 -9779.964,E2 -9779.964} C_VEL
LIN {X 0,Y 432.706,Z 380.443,A -85,B 0,C 180,E1 -9781.595,E2 -9781.595} C_VEL
LIN {X 0,Y 431.553,Z 395.549,A -85,B 0,C 180,E1 -9783.716,E2 -9783.716} C_VEL
LIN {X 0,Y 436.323,Z 423.881,A -85,B 0,C 180,E1 -9784.557,E2 -9784.557} C_VEL
LIN {X 0,Y 434.177,Z 563.487,A -85,B 0,C 180,E1 -9786.919,E2 -9786.919} C_VEL
LIN {X 0,Y 433.588,Z 578.523,A -85,B 0,C 180,E1 -9787.33,E2 -9787.33} C_VEL
LIN {X 0,Y 432.849,Z 592.282,A -85,B 0,C 180,E1 -9787.875,E2 -9787.875} C_VEL
LIN {X 0,Y 431.993,Z 606.888,A -85,B 0,C 180,E1 -9788.653,E2 -9788.653} C_VEL
LIN {X 0,Y 430.861,Z 620.824,A -85,B 0,C 180,E1 -9789.595,E2 -9789.595} C_VEL
LIN {X 0,Y 429.825,Z 633.553,A -85,B 0,C 180,E1 -9790.664,E2 -9790.664} C_VEL
LIN {X 0,Y 428.743,Z 645.307,A -85,B 0,C 180,E1 -9791.853,E2 -9791.853} C_VEL
LIN {X 0,Y 427.649,Z 657.071,A -85,B 0,C 180,E1 -9793.286,E2 -9793.286} C_VEL
LIN {X 0,Y 426.7,Z 666.952,A -85,B 0,C 180,E1 -9794.721,E2 -9794.721} C_VEL
LIN {X 0,Y 425.858,Z 676.595,A -85,B 0,C 180,E1 -9796.398,E2 -9796.398} C_VEL
LIN {X 0,Y 425.252,Z 684.612,A -85,B 0,C 180,E1 -9798.078,E2 -9798.078} C_VEL
LIN {X 0,Y 424.693,Z 692.075,A -85,B 0,C 180,E1 -9799.994,E2 -9799.994} C_VEL
LIN {X 0,Y 424.4,Z 697.992,A -85,B 0,C 180,E1 -9801.908,E2 -9801.908} C_VEL
LIN {X 0,Y 424.194,Z 702.403,A -85,B 0,C 180,E1 -9803.759,E2 -9803.759} C_VEL
LIN {X 0,Y 424.153,Z 705.024,A -85,B 0,C 180,E1 -9805.248,E2 -9805.248} C_VEL
LIN {X 0,Y 424.127,Z 707.355,A -85,B 0,C 180,E1 -9807.151,E2 -9807.151} C_VEL
LIN {X 0,Y 424.069,Z 708.528,A -85,B 0,C 180,E1 -9809.051,E2 -9809.051} C_VEL
LIN {X 0,Y 424.069,Z 708.528,A -85,B 0,C 180,E1 -9810.95,E2 -9810.95} C_VEL
LIN {X 0,Y 424.132,Z 707.357,A -85,B 0,C 180,E1 -9812.85,E2 -9812.85} C_VEL
LIN {X 0,Y 424.152,Z 705.023,A -85,B 0,C 180,E1 -9814.752,E2 -9814.752} C_VEL
LIN {X 0,Y 424.22,Z 701.473,A -85,B 0,C 180,E1 -9816.66,E2 -9816.66} C_VEL
LIN {X 0,Y 424.46,Z 696.622,A -85,B 0,C 180,E1 -9818.57,E2 -9818.57} C_VEL
LIN {X 0,Y 424.781,Z 690.344,A -85,B 0,C 180,E1 -9820.486,E2 -9820.486} C_VEL
LIN {X 0,Y 425.311,Z 683.556,A -85,B 0,C 180,E1 -9822.163,E2 -9822.163} C_VEL
LIN {X 0,Y 425.979,Z 675.34,A -85,B 0,C 180,E1 -9823.841,E2 -9823.841} C_VEL
LIN {X 0,Y 426.858,Z 665.429,A -85,B 0,C 180,E1 -9825.519,E2 -9825.519} C_VEL
LIN {X 0,Y 427.8,Z 655.263,A -85,B 0,C 180,E1 -9826.954,E2 -9826.954} C_VEL
LIN {X 0,Y 428.986,Z 643.124,A -85,B 0,C 180,E1 -9828.383,E2 -9828.383} C_VEL
LIN {X 0,Y 430.053,Z 630.928,A -85,B 0,C 180,E1 -9829.574,E2 -9829.574} C_VEL
LIN {X 0,Y 431.173,Z 617.622,A -85,B 0,C 180,E1 -9830.639,E2 -9830.639} C_VEL
LIN {X 0,Y 432.288,Z 602.845,A -85,B 0,C 180,E1 -9831.582,E2 -9831.582} C_VEL
LIN {X 0,Y 433.195,Z 587.723,A -85,B 0,C 180,E1 -9832.319,E2 -9832.319} C_VEL
LIN {X 0,Y 433.868,Z 572.594,A -85,B 0,C 180,E1 -9832.851,E2 -9832.851} C_VEL
LIN {X 0,Y 434.323,Z 557.169,A -85,B 0,C 180,E1 -9833.199,E2 -9833.199} C_VEL
LIN {X 0,Y 435.724,Z 470.922,A -85,B 0,C 180,E1 -9834.668,E2 -9834.668} C_VEL
LIN {X 0,Y 437.366,Z 423.399,A -85,B 0,C 180,E1 -9835.742,E2 -9835.742} C_VEL
LIN {X 0,Y 434.955,Z 407.01,A -85,B 0,C 180,E1 -9836.383,E2 -9836.383} C_VEL
LIN {X 0,Y 433.248,Z 398.473,A -85,B 0,C 180,E1 -9836.787,E2 -9836.787} C_VEL
LIN {X 0,Y 434.926,Z 386.063,A -85,B 0,C 180,E1 -9838.733,E2 -9838.733} C_VEL
LIN {X 0,Y 434.764,Z 383.519,A -85,B 0,C 180,E1 -9839.201,E2 -9839.201} C_VEL
LIN {X 0,Y 432.451,Z 373.67,A -85,B 0,C 180,E1 -9841.336,E2 -9841.336} C_VEL
LIN {X 0,Y 429.893,Z 365.11,A -85,B 0,C 180,E1 -9843.513,E2 -9843.513} C_VEL
LIN {X 0,Y 427.512,Z 358.419,A -85,B 0,C 180,E1 -9845.569,E2 -9845.569} C_VEL
LIN {X 0,Y 425.326,Z 352.277,A -85,B 0,C 180,E1 -9847.914,E2 -9847.914} C_VEL
LIN {X 0,Y 425.275,Z 352.138,A -85,B 0,C 180,E1 -9851.379,E2 -9851.379} C_VEL
LIN {X 0,Y 425.285,Z 352.137,A -85,B 0,C 180,E1 -9854.717,E2 -9854.717} C_VEL
LIN {X 0,Y 425.283,Z 352.137,A -85,B 0,C 180,E1 -9858.043,E2 -9858.043} C_VEL
LIN {X 0,Y 425.292,Z 352.136,A -85,B 0,C 180,E1 -9861.101,E2 -9861.101} C_VEL
LIN {X 0,Y 425.295,Z 352.364,A -85,B 0,C 180,E1 -9863.742,E2 -9863.742} C_VEL
LIN {X 0,Y 427.317,Z 357.846,A -85,B 0,C 180,E1 -9866,E2 -9866} C_VEL
LIN {X 0,Y 429.667,Z 365.273,A -85,B 0,C 180,E1 -9868.438,E2 -9868.438} C_VEL
LIN {X 0,Y 431.601,Z 372.486,A -85,B 0,C 180,E1 -9870.457,E2 -9870.457} C_VEL
LIN {X 0,Y 433.604,Z 381.799,A -85,B 0,C 180,E1 -9872.749,E2 -9872.749} C_VEL
LIN {X 0,Y 433.571,Z 384.418,A -85,B 0,C 180,E1 -9873.294,E2 -9873.294} C_VEL
LIN {X 0,Y 431.876,Z 398.63,A -85,B 0,C 180,E1 -9875.915,E2 -9875.915} C_VEL
LIN {X 0,Y 435.461,Z 414.542,A -85,B 0,C 180,E1 -9876.738,E2 -9876.738} C_VEL
LIN {X 0,Y 437.036,Z 424.563,A -85,B 0,C 180,E1 -9877.16,E2 -9877.16} C_VEL
LIN {X 0,Y 433.646,Z 505.765,A -85,B 0,C 180,E1 -9879.112,E2 -9879.112} C_VEL
LIN {X 0,Y 432.413,Z 543.352,A -85,B 0,C 180,E1 -9880.012,E2 -9880.012} C_VEL
LIN {X 0,Y 431.649,Z 558.18,A -85,B 0,C 180,E1 -9880.551,E2 -9880.551} C_VEL
LIN {X 0,Y 430.899,Z 573.262,A -85,B 0,C 180,E1 -9881.322,E2 -9881.322} C_VEL
LIN {X 0,Y 429.883,Z 587.524,A -85,B 0,C 180,E1 -9882.272,E2 -9882.272} C_VEL
LIN {X 0,Y 428.942,Z 600.227,A -85,B 0,C 180,E1 -9883.338,E2 -9883.338} C_VEL
LIN {X 0,Y 428.13,Z 611.818,A -85,B 0,C 180,E1 -9884.529,E2 -9884.529} C_VEL
LIN {X 0,Y 427.172,Z 623.17,A -85,B 0,C 180,E1 -9885.941,E2 -9885.941} C_VEL
LIN {X 0,Y 426.406,Z 632.687,A -85,B 0,C 180,E1 -9887.386,E2 -9887.386} C_VEL
LIN {X 0,Y 425.784,Z 640.508,A -85,B 0,C 180,E1 -9888.817,E2 -9888.817} C_VEL
LIN {X 0,Y 425.287,Z 647.955,A -85,B 0,C 180,E1 -9890.488,E2 -9890.488} C_VEL
LIN {X 0,Y 424.871,Z 653.157,A -85,B 0,C 180,E1 -9891.917,E2 -9891.917} C_VEL
LIN {X 0,Y 424.649,Z 657.312,A -85,B 0,C 180,E1 -9893.347,E2 -9893.347} C_VEL
LIN {X 0,Y 424.342,Z 661.486,A -85,B 0,C 180,E1 -9895.25,E2 -9895.25} C_VEL
LIN {X 0,Y 424.401,Z 662.997,A -85,B 0,C 180,E1 -9896.202,E2 -9896.202} C_VEL
LIN {X 0,Y 424.226,Z 664.95,A -85,B 0,C 180,E1 -9898.101,E2 -9898.101} C_VEL
LIN {X 0,Y 424.145,Z 665.463,A -85,B 0,C 180,E1 -9900,E2 -9900} C_VEL
LIN {X 0,Y 424.201,Z 664.559,A -85,B 0,C 180,E1 -9901.899,E2 -9901.899} C_VEL
LIN {X 0,Y 424.283,Z 663.578,A -85,B 0,C 180,E1 -9902.848,E2 -9902.848} C_VEL
LIN {X 0,Y 424.3,Z 660.537,A -85,B 0,C 180,E1 -9904.751,E2 -9904.751} C_VEL
LIN {X 0,Y 424.508,Z 656.873,A -85,B 0,C 180,E1 -9906.329,E2 -9906.329} C_VEL
LIN {X 0,Y 424.7,Z 651.471,A -85,B 0,C 180,E1 -9908.086,E2 -9908.086} C_VEL
LIN {X 0,Y 425.096,Z 644.903,A -85,B 0,C 180,E1 -9909.757,E2 -9909.757} C_VEL
LIN {X 0,Y 425.584,Z 636.719,A -85,B 0,C 180,E1 -9911.43,E2 -9911.43} C_VEL
LIN {X 0,Y 426.204,Z 628.168,A -85,B 0,C 180,E1 -9912.863,E2 -9912.863} C_VEL
LIN {X 0,Y 426.844,Z 617.866,A -85,B 0,C 180,E1 -9914.299,E2 -9914.299} C_VEL
LIN {X 0,Y 427.616,Z 606.402,A -85,B 0,C 180,E1 -9915.612,E2 -9915.612} C_VEL
LIN {X 0,Y 428.493,Z 593.593,A -85,B 0,C 180,E1 -9916.803,E2 -9916.803} C_VEL
LIN {X 0,Y 429.272,Z 580.971,A -85,B 0,C 180,E1 -9917.754,E2 -9917.754} C_VEL
LIN {X 0,Y 430.063,Z 566.568,A -85,B 0,C 180,E1 -9918.609,E2 -9918.609} C_VEL
LIN {X 0,Y 430.665,Z 551.846,A -85,B 0,C 180,E1 -9919.266,E2 -9919.266} C_VEL
LIN {X 0,Y 431.155,Z 537.375,A -85,B 0,C 180,E1 -9919.707,E2 -9919.707} C_VEL
LIN {X 0,Y 433.733,Z 422.943,A -85,B 0,C 180,E1 -9922.014,E2 -9922.014} C_VEL
LIN {X 0,Y 429.263,Z 397.866,A -85,B 0,C 180,E1 -9922.793,E2 -9922.793} C_VEL
LIN {X 0,Y 430.492,Z 380.729,A -85,B 0,C 180,E1 -9925.634,E2 -9925.634} C_VEL
LIN {X 0,Y 430.859,Z 376.416,A -85,B 0,C 180,E1 -9926.365,E2 -9926.365} C_VEL
LIN {X 0,Y 428.515,Z 365.683,A -85,B 0,C 180,E1 -9928.4,E2 -9928.4} C_VEL
LIN {X 0,Y 425.302,Z 352.46,A -85,B 0,C 180,E1 -9931.022,E2 -9931.022} C_VEL
LIN {X 0,Y 425.261,Z 352.141,A -85,B 0,C 180,E1 -9931.371,E2 -9931.371} C_VEL
LIN {X 0,Y 425.288,Z 352.137,A -85,B 0,C 180,E1 -9934.283,E2 -9934.283} C_VEL
LIN {X 0,Y 425.269,Z 352.138,A -85,B 0,C 180,E1 -9937.695,E2 -9937.695} C_VEL
LIN {X 0,Y 425.241,Z 352.139,A -85,B 0,C 180,E1 -9940.514,E2 -9940.514} C_VEL
LIN {X 0,Y 425.244,Z 352.128,A -85,B 0,C 180,E1 -9943.349,E2 -9943.349} C_VEL
LIN {X 0,Y 425.255,Z 352.131,A -85,B 0,C 180,E1 -9946.043,E2 -9946.043} C_VEL
LIN {X 0,Y 425.245,Z 352.141,A -85,B 0,C 180,E1 -9948.618,E2 -9948.618} C_VEL
LIN {X 0,Y 425.269,Z 352.136,A -85,B 0,C 180,E1 -9952.304,E2 -9952.304} C_VEL
LIN {X 0,Y 425.282,Z 352.131,A -85,B 0,C 180,E1 -9955.815,E2 -9955.815} C_VEL
LIN {X 0,Y 425.321,Z 352.397,A -85,B 0,C 180,E1 -9956.566,E2 -9956.566} C_VEL
LIN {X 0,Y 429.583,Z 368.282,A -85,B 0,C 180,E1 -9959.299,E2 -9959.299} C_VEL
LIN {X 0,Y 432.276,Z 379.918,A -85,B 0,C 180,E1 -9961.199,E2 -9961.199} C_VEL
LIN {X 0,Y 431.498,Z 397.119,A -85,B 0,C 180,E1 -9963.53,E2 -9963.53} C_VEL
LIN {X 0,Y 436.987,Z 425.671,A -85,B 0,C 180,E1 -9964.414,E2 -9964.414} C_VEL
LIN {X 0,Y 436.461,Z 463.211,A -85,B 0,C 180,E1 -9965.052,E2 -9965.052} C_VEL
LIN {X 0,Y 435.846,Z 469.057,A -85,B 0,C 180,E1 -9965.119,E2 -9965.119} C_VEL
LIN {X 0,Y 430.288,Z 488.115,A -85,B 0,C 180,E1 -9965.122,E2 -9965.122} C_VEL
LIN {X 0,Y 429.547,Z 493.97,A -85,B 0,C 180,E1 -9965.182,E2 -9965.182} C_VEL
LIN {X 0,Y 428.258,Z 565.172,A -85,B 0,C 180,E1 -9966.421,E2 -9966.421} C_VEL
LIN {X 0,Y 427.594,Z 580.526,A -85,B 0,C 180,E1 -9966.867,E2 -9966.867} C_VEL
LIN {X 0,Y 426.814,Z 594.299,A -85,B 0,C 180,E1 -9967.442,E2 -9967.442} C_VEL
LIN {X 0,Y 425.85,Z 608.195,A -85,B 0,C 180,E1 -9968.202,E2 -9968.202} C_VEL
LIN {X 0,Y 424.671,Z 621.994,A -85,B 0,C 180,E1 -9969.157,E2 -9969.157} C_VEL
LIN {X 0,Y 423.337,Z 635.909,A -85,B 0,C 180,E1 -9970.356,E2 -9970.356} C_VEL
LIN {X 0,Y 422.116,Z 647.994,A -85,B 0,C 180,E1 -9971.626,E2 -9971.626} C_VEL
LIN {X 0,Y 420.991,Z 659.015,A -85,B 0,C 180,E1 -9973.013,E2 -9973.013} C_VEL
LIN {X 0,Y 420.019,Z 668.776,A -85,B 0,C 180,E1 -9974.471,E2 -9974.471} C_VEL
LIN {X 0,Y 419.035,Z 678.326,A -85,B 0,C 180,E1 -9976.172,E2 -9976.172} C_VEL
LIN {X 0,Y 418.389,Z 686.286,A -85,B 0,C 180,E1 -9977.879,E2 -9977.879} C_VEL
LIN {X 0,Y 417.718,Z 693.699,A -85,B 0,C 180,E1 -9979.825,E2 -9979.825} C_VEL
LIN {X 0,Y 417.361,Z 699.585,A -85,B 0,C 180,E1 -9981.771,E2 -9981.771} C_VEL
LIN {X 0,Y 417.105,Z 704.238,A -85,B 0,C 180,E1 -9983.784,E2 -9983.784} C_VEL
LIN {X 0,Y 417.058,Z 706.611,A -85,B 0,C 180,E1 -9985.167,E2 -9985.167} C_VEL
LIN {X 0,Y 416.975,Z 708.954,A -85,B 0,C 180,E1 -9987.102,E2 -9987.102} C_VEL
LIN {X 0,Y 416.99,Z 710.146,A -85,B 0,C 180,E1 -9989.034,E2 -9989.034} C_VEL
LIN {X 0,Y 416.991,Z 710.161,A -85,B 0,C 180,E1 -9990.966,E2 -9990.966} C_VEL
LIN {X 0,Y 416.976,Z 709.027,A -85,B 0,C 180,E1 -9992.898,E2 -9992.898} C_VEL
LIN {X 0,Y 417.063,Z 706.746,A -85,B 0,C 180,E1 -9994.833,E2 -9994.833} C_VEL
LIN {X 0,Y 417.226,Z 703.267,A -85,B 0,C 180,E1 -9996.772,E2 -9996.772} C_VEL
LIN {X 0,Y 417.419,Z 698.502,A -85,B 0,C 180,E1 -9998.716,E2 -9998.716} C_VEL
LIN {X 0,Y 417.804,Z 692.322,A -85,B 0,C 180,E1 -10000.663,E2 -10000.663} C_VEL
LIN {X 0,Y 418.401,Z 685.653,A -85,B 0,C 180,E1 -10002.366,E2 -10002.366} C_VEL
LIN {X 0,Y 419.113,Z 677.575,A -85,B 0,C 180,E1 -10004.072,E2 -10004.072} C_VEL
LIN {X 0,Y 420.115,Z 667.871,A -85,B 0,C 180,E1 -10005.774,E2 -10005.774} C_VEL
LIN {X 0,Y 421.162,Z 657.93,A -85,B 0,C 180,E1 -10007.229,E2 -10007.229} C_VEL
LIN {X 0,Y 422.347,Z 646.131,A -85,B 0,C 180,E1 -10008.683,E2 -10008.683} C_VEL
LIN {X 0,Y 423.532,Z 634.345,A -85,B 0,C 180,E1 -10009.887,E2 -10009.887} C_VEL
LIN {X 0,Y 424.701,Z 621.609,A -85,B 0,C 180,E1 -10010.968,E2 -10010.968} C_VEL
LIN {X 0,Y 425.874,Z 607.717,A -85,B 0,C 180,E1 -10011.923,E2 -10011.923} C_VEL
LIN {X 0,Y 426.847,Z 593.747,A -85,B 0,C 180,E1 -10012.681,E2 -10012.681} C_VEL
LIN {X 0,Y 427.64,Z 579.59,A -85,B 0,C 180,E1 -10013.262,E2 -10013.262} C_VEL
LIN {X 0,Y 428.285,Z 563.817,A -85,B 0,C 180,E1 -10013.705,E2 -10013.705} C_VEL
LIN {X 0,Y 430.662,Z 428.077,A -85,B 0,C 180,E1 -10016.04,E2 -10016.04} C_VEL
LIN {X 0,Y 428.57,Z 415.729,A -85,B 0,C 180,E1 -10016.402,E2 -10016.402} C_VEL
LIN {X 0,Y 424.818,Z 396.863,A -85,B 0,C 180,E1 -10017.032,E2 -10017.032} C_VEL
LIN {X 0,Y 425.578,Z 382.991,A -85,B 0,C 180,E1 -10018.926,E2 -10018.926} C_VEL
LIN {X 0,Y 424.704,Z 377.679,A -85,B 0,C 180,E1 -10019.765,E2 -10019.765} C_VEL
LIN {X 0,Y 420.947,Z 362.712,A -85,B 0,C 180,E1 -10022.294,E2 -10022.294} C_VEL
LIN {X 0,Y 418.278,Z 353.177,A -85,B 0,C 180,E1 -10024,E2 -10024} C_VEL
LIN {X 0,Y 418.231,Z 353.014,A -85,B 0,C 180,E1 -10027.225,E2 -10027.225} C_VEL
LIN {X 0,Y 418.205,Z 353.015,A -85,B 0,C 180,E1 -10030.95,E2 -10030.95} C_VEL
LIN {X 0,Y 418.202,Z 353.019,A -85,B 0,C 180,E1 -10033.728,E2 -10033.728} C_VEL
LIN {X 0,Y 418.199,Z 353.019,A -85,B 0,C 180,E1 -10036.447,E2 -10036.447} C_VEL
LIN {X 0,Y 418.206,Z 353.017,A -85,B 0,C 180,E1 -10039.133,E2 -10039.133} C_VEL
LIN {X 0,Y 418.234,Z 353.012,A -85,B 0,C 180,E1 -10042.775,E2 -10042.775} C_VEL
LIN {X 0,Y 418.237,Z 353.012,A -85,B 0,C 180,E1 -10046.322,E2 -10046.322} C_VEL
LIN {X 0,Y 418.242,Z 353.01,A -85,B 0,C 180,E1 -10049.728,E2 -10049.728} C_VEL
LIN {X 0,Y 418.226,Z 353.002,A -85,B 0,C 180,E1 -10053.018,E2 -10053.018} C_VEL
LIN {X 0,Y 418.259,Z 353.005,A -85,B 0,C 180,E1 -10056.217,E2 -10056.217} C_VEL
LIN {X 0,Y 418.25,Z 353.006,A -85,B 0,C 180,E1 -10059.337,E2 -10059.337} C_VEL
LIN {X 0,Y 418.28,Z 352.996,A -85,B 0,C 180,E1 -10062.396,E2 -10062.396} C_VEL
LIN {X 0,Y 418.303,Z 353.003,A -85,B 0,C 180,E1 -10065.403,E2 -10065.403} C_VEL
LIN {X 0,Y 418.314,Z 352.99,A -85,B 0,C 180,E1 -10068.369,E2 -10068.369} C_VEL
LIN {X 0,Y 418.466,Z 352.981,A -85,B 0,C 180,E1 -10072.278,E2 -10072.278} C_VEL
LIN {X 0,Y 418.509,Z 352.966,A -85,B 0,C 180,E1 -10074.217,E2 -10074.217} C_VEL
LIN {X 0,Y 418.539,Z 352.973,A -85,B 0,C 180,E1 -10078.075,E2 -10078.075} C_VEL
LIN {X 0,Y 418.669,Z 352.95,A -85,B 0,C 180,E1 -10080,E2 -10080} C_VEL
LIN {X 0,Y 418.495,Z 352.97,A -85,B 0,C 180,E1 -10082.888,E2 -10082.888} C_VEL
LIN {X 0,Y 418.5,Z 352.974,A -85,B 0,C 180,E1 -10085.783,E2 -10085.783} C_VEL
LIN {X 0,Y 418.378,Z 352.98,A -85,B 0,C 180,E1 -10088.695,E2 -10088.695} C_VEL
LIN {X 0,Y 418.316,Z 352.998,A -85,B 0,C 180,E1 -10091.631,E2 -10091.631} C_VEL
LIN {X 0,Y 418.303,Z 352.99,A -85,B 0,C 180,E1 -10094.597,E2 -10094.597} C_VEL
LIN {X 0,Y 418.28,Z 353.003,A -85,B 0,C 180,E1 -10097.604,E2 -10097.604} C_VEL
LIN {X 0,Y 418.25,Z 353.001,A -85,B 0,C 180,E1 -10100.663,E2 -10100.663} C_VEL
LIN {X 0,Y 418.287,Z 352.999,A -85,B 0,C 180,E1 -10103.781,E2 -10103.781} C_VEL
LIN {X 0,Y 418.31,Z 353.004,A -85,B 0,C 180,E1 -10107.07,E2 -10107.07} C_VEL
LIN {X 0,Y 418.245,Z 353,A -85,B 0,C 180,E1 -10110.272,E2 -10110.272} C_VEL
LIN {X 0,Y 418.248,Z 353.003,A -85,B 0,C 180,E1 -10113.677,E2 -10113.677} C_VEL
LIN {X 0,Y 418.239,Z 353.01,A -85,B 0,C 180,E1 -10117.224,E2 -10117.224} C_VEL
LIN {X 0,Y 418.244,Z 352.979,A -85,B 0,C 180,E1 -10119.683,E2 -10119.683} C_VEL
LIN {X 0,Y 418.232,Z 353.005,A -85,B 0,C 180,E1 -10122.321,E2 -10122.321} C_VEL
LIN {X 0,Y 418.238,Z 353.002,A -85,B 0,C 180,E1 -10125.109,E2 -10125.109} C_VEL
LIN {X 0,Y 418.24,Z 352.995,A -85,B 0,C 180,E1 -10127.767,E2 -10127.767} C_VEL
LIN {X 0,Y 418.255,Z 353.013,A -85,B 0,C 180,E1 -10130.619,E2 -10130.619} C_VEL
LIN {X 0,Y 418.243,Z 353.011,A -85,B 0,C 180,E1 -10133.976,E2 -10133.976} C_VEL
LIN {X 0,Y 418.316,Z 353.197,A -85,B 0,C 180,E1 -10136.414,E2 -10136.414} C_VEL
LIN {X 0,Y 423.307,Z 371.745,A -85,B 0,C 180,E1 -10139.693,E2 -10139.693} C_VEL
LIN {X 0,Y 425.838,Z 381.974,A -85,B 0,C 180,E1 -10141.405,E2 -10141.405} C_VEL
LIN {X 0,Y 425.564,Z 387.359,A -85,B 0,C 180,E1 -10142.19,E2 -10142.19} C_VEL
LIN {X 0,Y 424.89,Z 395.231,A -85,B 0,C 180,E1 -10143.278,E2 -10143.278} C_VEL
LIN {X 0,Y 429.836,Z 424.372,A -85,B 0,C 180,E1 -10144.151,E2 -10144.151} C_VEL
LIN {X 0,Y 429.066,Z 480.533,A -85,B 0,C 180,E1 -10145.118,E2 -10145.118} C_VEL
LIN {X 0,Y 427.611,Z 565.087,A -85,B 0,C 180,E1 -10146.576,E2 -10146.576} C_VEL
LIN {X 0,Y 426.989,Z 580.663,A -85,B 0,C 180,E1 -10147.033,E2 -10147.033} C_VEL
LIN {X 0,Y 426.213,Z 594.359,A -85,B 0,C 180,E1 -10147.612,E2 -10147.612} C_VEL
LIN {X 0,Y 425.234,Z 608.903,A -85,B 0,C 180,E1 -10148.424,E2 -10148.424} C_VEL
LIN {X 0,Y 424.07,Z 622.433,A -85,B 0,C 180,E1 -10149.38,E2 -10149.38} C_VEL
LIN {X 0,Y 422.829,Z 636.154,A -85,B 0,C 180,E1 -10150.584,E2 -10150.584} C_VEL
LIN {X 0,Y 421.623,Z 648.535,A -85,B 0,C 180,E1 -10151.914,E2 -10151.914} C_VEL
LIN {X 0,Y 420.429,Z 660.617,A -85,B 0,C 180,E1 -10153.49,E2 -10153.49} C_VEL
LIN {X 0,Y 419.397,Z 671.344,A -85,B 0,C 180,E1 -10155.194,E2 -10155.194} C_VEL
LIN {X 0,Y 418.559,Z 680.14,A -85,B 0,C 180,E1 -10156.874,E2 -10156.874} C_VEL
LIN {X 0,Y 417.942,Z 688.566,A -85,B 0,C 180,E1 -10158.85,E2 -10158.85} C_VEL
LIN {X 0,Y 417.464,Z 695.232,A -85,B 0,C 180,E1 -10160.797,E2 -10160.797} C_VEL
LIN {X 0,Y 417.236,Z 700.436,A -85,B 0,C 180,E1 -10162.742,E2 -10162.742} C_VEL
LIN {X 0,Y 417.082,Z 703.424,A -85,B 0,C 180,E1 -10164.197,E2 -10164.197} C_VEL
LIN {X 0,Y 416.984,Z 706.351,A -85,B 0,C 180,E1 -10166.134,E2 -10166.134} C_VEL
LIN {X 0,Y 417.069,Z 708.098,A -85,B 0,C 180,E1 -10168.069,E2 -10168.069} C_VEL
LIN {X 0,Y 416.961,Z 708.695,A -85,B 0,C 180,E1 -10170,E2 -10170} C_VEL
LIN {X 0,Y 417.071,Z 708.099,A -85,B 0,C 180,E1 -10171.931,E2 -10171.931} C_VEL
LIN {X 0,Y 416.984,Z 706.352,A -85,B 0,C 180,E1 -10173.866,E2 -10173.866} C_VEL
LIN {X 0,Y 417.077,Z 703.419,A -85,B 0,C 180,E1 -10175.803,E2 -10175.803} C_VEL
LIN {X 0,Y 417.281,Z 699.231,A -85,B 0,C 180,E1 -10177.744,E2 -10177.744} C_VEL
LIN {X 0,Y 417.57,Z 693.686,A -85,B 0,C 180,E1 -10179.69,E2 -10179.69} C_VEL
LIN {X 0,Y 418.116,Z 686.626,A -85,B 0,C 180,E1 -10181.637,E2 -10181.637} C_VEL
LIN {X 0,Y 418.649,Z 679.492,A -85,B 0,C 180,E1 -10183.256,E2 -10183.256} C_VEL
LIN {X 0,Y 419.548,Z 669.903,A -85,B 0,C 180,E1 -10185.049,E2 -10185.049} C_VEL
LIN {X 0,Y 420.406,Z 660.585,A -85,B 0,C 180,E1 -10186.511,E2 -10186.511} C_VEL
LIN {X 0,Y 421.597,Z 649.103,A -85,B 0,C 180,E1 -10188.013,E2 -10188.013} C_VEL
LIN {X 0,Y 422.738,Z 637.323,A -85,B 0,C 180,E1 -10189.294,E2 -10189.294} C_VEL
LIN {X 0,Y 423.998,Z 623.916,A -85,B 0,C 180,E1 -10190.497,E2 -10190.497} C_VEL
LIN {X 0,Y 425.093,Z 610.708,A -85,B 0,C 180,E1 -10191.456,E2 -10191.456} C_VEL
LIN {X 0,Y 426.121,Z 596.172,A -85,B 0,C 180,E1 -10192.293,E2 -10192.293} C_VEL
LIN {X 0,Y 427.008,Z 580.869,A -85,B 0,C 180,E1 -10192.952,E2 -10192.952} C_VEL
LIN {X 0,Y 427.592,Z 566.114,A -85,B 0,C 180,E1 -10193.393,E2 -10193.393} C_VEL
LIN {X 0,Y 428.61,Z 507.077,A -85,B 0,C 180,E1 -10194.426,E2 -10194.426} C_VEL
LIN {X 0,Y 429.141,Z 481.939,A -85,B 0,C 180,E1 -10194.878,E2 -10194.878} C_VEL
LIN {X 0,Y 431.287,Z 424.503,A -85,B 0,C 180,E1 -10196.216,E2 -10196.216} C_VEL
LIN {X 0,Y 429.177,Z 409.47,A -85,B 0,C 180,E1 -10196.82,E2 -10196.82} C_VEL
LIN {X 0,Y 427.05,Z 398.473,A -85,B 0,C 180,E1 -10197.375,E2 -10197.375} C_VEL
LIN {X 0,Y 428.407,Z 389.045,A -85,B 0,C 180,E1 -10198.889,E2 -10198.889} C_VEL
LIN {X 0,Y 428.544,Z 387.152,A -85,B 0,C 180,E1 -10199.225,E2 -10199.225} C_VEL
LIN {X 0,Y 426.476,Z 377.727,A -85,B 0,C 180,E1 -10201.293,E2 -10201.293} C_VEL
LIN {X 0,Y 423.996,Z 369.125,A -85,B 0,C 180,E1 -10203.53,E2 -10203.53} C_VEL
LIN {X 0,Y 421.622,Z 362.274,A -85,B 0,C 180,E1 -10205.691,E2 -10205.691} C_VEL
LIN {X 0,Y 419.486,Z 356.258,A -85,B 0,C 180,E1 -10208.054,E2 -10208.054} C_VEL
LIN {X 0,Y 418.259,Z 353.093,A -85,B 0,C 180,E1 -10209.755,E2 -10209.755} C_VEL
LIN {X 0,Y 418.23,Z 353.016,A -85,B 0,C 180,E1 -10212.321,E2 -10212.321} C_VEL
LIN {X 0,Y 418.236,Z 353.015,A -85,B 0,C 180,E1 -10215.109,E2 -10215.109} C_VEL
LIN {X 0,Y 418.235,Z 353.016,A -85,B 0,C 180,E1 -10217.766,E2 -10217.766} C_VEL
LIN {X 0,Y 418.242,Z 353.015,A -85,B 0,C 180,E1 -10220.621,E2 -10220.621} C_VEL
LIN {X 0,Y 418.251,Z 353.239,A -85,B 0,C 180,E1 -10221.991,E2 -10221.991} C_VEL
LIN {X 0,Y 419.761,Z 357.347,A -85,B 0,C 180,E1 -10224.126,E2 -10224.126} C_VEL
LIN {X 0,Y 421.989,Z 363.696,A -85,B 0,C 180,E1 -10226.661,E2 -10226.661} C_VEL
LIN {X 0,Y 424.237,Z 371.281,A -85,B 0,C 180,E1 -10229.099,E2 -10229.099} C_VEL
LIN {X 0,Y 426.296,Z 379.886,A -85,B 0,C 180,E1 -10231.439,E2 -10231.439} C_VEL
LIN {X 0,Y 427.236,Z 384.889,A -85,B 0,C 180,E1 -10232.66,E2 -10232.66} C_VEL
LIN {X 0,Y 426.307,Z 392.148,A -85,B 0,C 180,E1 -10234.096,E2 -10234.096} C_VEL
LIN {X 0,Y 425.566,Z 398.772,A -85,B 0,C 180,E1 -10235.312,E2 -10235.312} C_VEL
LIN {X 0,Y 428.997,Z 413.626,A -85,B 0,C 180,E1 -10236.136,E2 -10236.136} C_VEL
LIN {X 0,Y 430.966,Z 424.911,A -85,B 0,C 180,E1 -10236.657,E2 -10236.657} C_VEL
LIN {X 0,Y 427.449,Z 502.762,A -85,B 0,C 180,E1 -10238.605,E2 -10238.605} C_VEL
LIN {X 0,Y 425.95,Z 544.128,A -85,B 0,C 180,E1 -10239.633,E2 -10239.633} C_VEL
LIN {X 0,Y 425.167,Z 558.543,A -85,B 0,C 180,E1 -10240.174,E2 -10240.174} C_VEL
LIN {X 0,Y 424.394,Z 572.786,A -85,B 0,C 180,E1 -10240.911,E2 -10240.911} C_VEL
LIN {X 0,Y 423.495,Z 585.462,A -85,B 0,C 180,E1 -10241.746,E2 -10241.746} C_VEL
LIN {X 0,Y 422.422,Z 598.583,A -85,B 0,C 180,E1 -10242.824,E2 -10242.824} C_VEL
LIN {X 0,Y 421.539,Z 610.476,A -85,B 0,C 180,E1 -10244.033,E2 -10244.033} C_VEL
LIN {X 0,Y 420.469,Z 622.201,A -85,B 0,C 180,E1 -10245.48,E2 -10245.48} C_VEL
LIN {X 0,Y 419.625,Z 631.866,A -85,B 0,C 180,E1 -10246.932,E2 -10246.932} C_VEL
LIN {X 0,Y 418.835,Z 641.094,A -85,B 0,C 180,E1 -10248.629,E2 -10248.629} C_VEL
LIN {X 0,Y 418.307,Z 648.5,A -85,B 0,C 180,E1 -10250.328,E2 -10250.328} C_VEL
LIN {X 0,Y 417.863,Z 653.68,A -85,B 0,C 180,E1 -10251.781,E2 -10251.781} C_VEL
LIN {X 0,Y 417.597,Z 658.563,A -85,B 0,C 180,E1 -10253.532,E2 -10253.532} C_VEL
LIN {X 0,Y 417.275,Z 661.947,A -85,B 0,C 180,E1 -10255.169,E2 -10255.169} C_VEL
LIN {X 0,Y 417.343,Z 663.438,A -85,B 0,C 180,E1 -10256.138,E2 -10256.138} C_VEL
LIN {X 0,Y 417.151,Z 665.344,A -85,B 0,C 180,E1 -10258.069,E2 -10258.069} C_VEL
LIN {X 0,Y 417.062,Z 665.81,A -85,B 0,C 180,E1 -10260,E2 -10260} C_VEL
LIN {X 0,Y 417.127,Z 664.859,A -85,B 0,C 180,E1 -10261.931,E2 -10261.931} C_VEL
LIN {X 0,Y 417.216,Z 663.852,A -85,B 0,C 180,E1 -10262.897,E2 -10262.897} C_VEL
LIN {X 0,Y 417.236,Z 660.754,A -85,B 0,C 180,E1 -10264.831,E2 -10264.831} C_VEL
LIN {X 0,Y 417.477,Z 656.128,A -85,B 0,C 180,E1 -10266.768,E2 -10266.768} C_VEL
LIN {X 0,Y 417.639,Z 651.558,A -85,B 0,C 180,E1 -10268.224,E2 -10268.224} C_VEL
LIN {X 0,Y 418.05,Z 644.912,A -85,B 0,C 180,E1 -10269.923,E2 -10269.923} C_VEL
LIN {X 0,Y 418.585,Z 636.639,A -85,B 0,C 180,E1 -10271.624,E2 -10271.624} C_VEL
LIN {X 0,Y 419.245,Z 627.076,A -85,B 0,C 180,E1 -10273.225,E2 -10273.225} C_VEL
LIN {X 0,Y 419.891,Z 617.572,A -85,B 0,C 180,E1 -10274.541,E2 -10274.541} C_VEL
LIN {X 0,Y 420.739,Z 605.925,A -85,B 0,C 180,E1 -10275.874,E2 -10275.874} C_VEL
LIN {X 0,Y 421.543,Z 594.394,A -85,B 0,C 180,E1 -10276.964,E2 -10276.964} C_VEL
LIN {X 0,Y 422.349,Z 581.896,A -85,B 0,C 180,E1 -10277.93,E2 -10277.93} C_VEL
LIN {X 0,Y 423.128,Z 567.998,A -85,B 0,C 180,E1 -10278.782,E2 -10278.782} C_VEL
LIN {X 0,Y 423.753,Z 554.035,A -85,B 0,C 180,E1 -10279.435,E2 -10279.435} C_VEL
LIN {X 0,Y 424.268,Z 539.661,A -85,B 0,C 180,E1 -10279.915,E2 -10279.915} C_VEL
LIN {X 0,Y 427.025,Z 423.379,A -85,B 0,C 180,E1 -10282.332,E2 -10282.332} C_VEL
LIN {X 0,Y 422.456,Z 397.86,A -85,B 0,C 180,E1 -10283.146,E2 -10283.146} C_VEL
LIN {X 0,Y 423.937,Z 379.051,A -85,B 0,C 180,E1 -10286.317,E2 -10286.317} C_VEL
LIN {X 0,Y 423.342,Z 374.478,A -85,B 0,C 180,E1 -10287.164,E2 -10287.164} C_VEL
LIN {X 0,Y 419.403,Z 357.907,A -85,B 0,C 180,E1 -10290.423,E2 -10290.423} C_VEL
LIN {X 0,Y 418.264,Z 353.26,A -85,B 0,C 180,E1 -10291.392,E2 -10291.392} C_VEL
LIN {X 0,Y 418.242,Z 353.014,A -85,B 0,C 180,E1 -10292.84,E2 -10292.84} C_VEL
LIN {X 0,Y 418.238,Z 353.015,A -85,B 0,C 180,E1 -10296.236,E2 -10296.236} C_VEL
LIN {X 0,Y 418.198,Z 353.019,A -85,B 0,C 180,E1 -10299.688,E2 -10299.688} C_VEL
LIN {X 0,Y 418.206,Z 353.001,A -85,B 0,C 180,E1 -10302.317,E2 -10302.317} C_VEL
LIN {X 0,Y 418.235,Z 353.013,A -85,B 0,C 180,E1 -10305.108,E2 -10305.108} C_VEL
LIN {X 0,Y 418.217,Z 353.006,A -85,B 0,C 180,E1 -10307.764,E2 -10307.764} C_VEL
LIN {X 0,Y 418.227,Z 353.012,A -85,B 0,C 180,E1 -10311.555,E2 -10311.555} C_VEL
LIN {X 0,Y 418.248,Z 353.008,A -85,B 0,C 180,E1 -10315.158,E2 -10315.158} C_VEL
LIN {X 0,Y 418.279,Z 353.255,A -85,B 0,C 180,E1 -10316.126,E2 -10316.126} C_VEL
LIN {X 0,Y 422.396,Z 368.4,A -85,B 0,C 180,E1 -10318.785,E2 -10318.785} C_VEL
LIN {X 0,Y 425.308,Z 380.34,A -85,B 0,C 180,E1 -10320.774,E2 -10320.774} C_VEL
LIN {X 0,Y 425.534,Z 383.711,A -85,B 0,C 180,E1 -10321.28,E2 -10321.28} C_VEL
LIN {X 0,Y 424.882,Z 397.148,A -85,B 0,C 180,E1 -10323.092,E2 -10323.092} C_VEL
LIN {X 0,Y 430.555,Z 426.756,A -85,B 0,C 180,E1 -10324.025,E2 -10324.025} C_VEL
LIN {X 0,Y 429.547,Z 493.97,A -85,B 0,C 180,E1 -10325.182,E2 -10325.182} C_VEL
LIN {X 0,Y 428.809,Z 499.823,A -85,B 0,C 180,E1 -10325.243,E2 -10325.243} C_VEL
LIN {X 0,Y 423.215,Z 518.871,A -85,B 0,C 180,E1 -10325.245,E2 -10325.245} C_VEL
LIN {X 0,Y 422.557,Z 524.719,A -85,B 0,C 180,E1 -10325.312,E2 -10325.312} C_VEL
LIN {X 0,Y 421.764,Z 565.088,A -85,B 0,C 180,E1 -10326.035,E2 -10326.035} C_VEL
LIN {X 0,Y 421.084,Z 580.096,A -85,B 0,C 180,E1 -10326.473,E2 -10326.473} C_VEL
LIN {X 0,Y 420.29,Z 593.552,A -85,B 0,C 180,E1 -10327.035,E2 -10327.035} C_VEL
LIN {X 0,Y 419.248,Z 608.164,A -85,B 0,C 180,E1 -10327.841,E2 -10327.841} C_VEL
LIN {X 0,Y 418.019,Z 621.968,A -85,B 0,C 180,E1 -10328.809,E2 -10328.809} C_VEL
LIN {X 0,Y 416.632,Z 635.887,A -85,B 0,C 180,E1 -10330.026,E2 -10330.026} C_VEL
LIN {X 0,Y 415.282,Z 648.609,A -85,B 0,C 180,E1 -10331.39,E2 -10331.39} C_VEL
LIN {X 0,Y 414.159,Z 658.997,A -85,B 0,C 180,E1 -10332.725,E2 -10332.725} C_VEL
LIN {X 0,Y 413.123,Z 668.759,A -85,B 0,C 180,E1 -10334.205,E2 -10334.205} C_VEL
LIN {X 0,Y 412.089,Z 678.31,A -85,B 0,C 180,E1 -10335.935,E2 -10335.935} C_VEL
LIN {X 0,Y 411.38,Z 686.271,A -85,B 0,C 180,E1 -10337.669,E2 -10337.669} C_VEL
LIN {X 0,Y 410.689,Z 693.685,A -85,B 0,C 180,E1 -10339.649,E2 -10339.649} C_VEL
LIN {X 0,Y 410.292,Z 699.571,A -85,B 0,C 180,E1 -10341.628,E2 -10341.628} C_VEL
LIN {X 0,Y 410.076,Z 703.049,A -85,B 0,C 180,E1 -10343.11,E2 -10343.11} C_VEL
LIN {X 0,Y 409.967,Z 706.598,A -85,B 0,C 180,E1 -10345.083,E2 -10345.083} C_VEL
LIN {X 0,Y 409.873,Z 708.941,A -85,B 0,C 180,E1 -10347.051,E2 -10347.051} C_VEL
LIN {X 0,Y 409.916,Z 710.132,A -85,B 0,C 180,E1 -10349.017,E2 -10349.017} C_VEL
LIN {X 0,Y 409.916,Z 710.147,A -85,B 0,C 180,E1 -10350.982,E2 -10350.982} C_VEL
LIN {X 0,Y 409.874,Z 709.013,A -85,B 0,C 180,E1 -10352.948,E2 -10352.948} C_VEL
LIN {X 0,Y 409.974,Z 706.731,A -85,B 0,C 180,E1 -10354.917,E2 -10354.917} C_VEL
LIN {X 0,Y 410.157,Z 703.252,A -85,B 0,C 180,E1 -10356.889,E2 -10356.889} C_VEL
LIN {X 0,Y 410.373,Z 698.485,A -85,B 0,C 180,E1 -10358.866,E2 -10358.866} C_VEL
LIN {X 0,Y 410.789,Z 692.304,A -85,B 0,C 180,E1 -10360.847,E2 -10360.847} C_VEL
LIN {X 0,Y 411.384,Z 685.634,A -85,B 0,C 180,E1 -10362.581,E2 -10362.581} C_VEL
LIN {X 0,Y 412.181,Z 677.554,A -85,B 0,C 180,E1 -10364.314,E2 -10364.314} C_VEL
LIN {X 0,Y 413.223,Z 667.849,A -85,B 0,C 180,E1 -10366.044,E2 -10366.044} C_VEL
LIN {X 0,Y 414.341,Z 657.905,A -85,B 0,C 180,E1 -10367.522,E2 -10367.522} C_VEL
LIN {X 0,Y 415.569,Z 646.103,A -85,B 0,C 180,E1 -10368.999,E2 -10368.999} C_VEL
LIN {X 0,Y 416.834,Z 634.314,A -85,B 0,C 180,E1 -10370.221,E2 -10370.221} C_VEL
LIN {X 0,Y 418.06,Z 621.572,A -85,B 0,C 180,E1 -10371.318,E2 -10371.318} C_VEL
LIN {X 0,Y 419.286,Z 607.671,A -85,B 0,C 180,E1 -10372.286,E2 -10372.286} C_VEL
LIN {X 0,Y 420.263,Z 593.689,A -85,B 0,C 180,E1 -10373.057,E2 -10373.057} C_VEL
LIN {X 0,Y 421.144,Z 578.65,A -85,B 0,C 180,E1 -10373.675,E2 -10373.675} C_VEL
LIN {X 0,Y 421.788,Z 563.692,A -85,B 0,C 180,E1 -10374.094,E2 -10374.094} C_VEL
LIN {X 0,Y 424.291,Z 429.265,A -85,B 0,C 180,E1 -10376.436,E2 -10376.436} C_VEL
LIN {X 0,Y 422.658,Z 419.071,A -85,B 0,C 180,E1 -10376.736,E2 -10376.736} C_VEL
LIN {X 0,Y 418.248,Z 396.979,A -85,B 0,C 180,E1 -10377.475,E2 -10377.475} C_VEL
LIN {X 0,Y 418.87,Z 384.068,A -85,B 0,C 180,E1 -10379.252,E2 -10379.252} C_VEL
LIN {X 0,Y 416.065,Z 371.647,A -85,B 0,C 180,E1 -10381.313,E2 -10381.313} C_VEL
LIN {X 0,Y 411.976,Z 356.729,A -85,B 0,C 180,E1 -10383.939,E2 -10383.939} C_VEL
LIN {X 0,Y 411.225,Z 353.964,A -85,B 0,C 180,E1 -10384.501,E2 -10384.501} C_VEL
LIN {X 0,Y 411.185,Z 353.891,A -85,B 0,C 180,E1 -10388.165,E2 -10388.165} C_VEL
LIN {X 0,Y 411.158,Z 353.896,A -85,B 0,C 180,E1 -10391.808,E2 -10391.808} C_VEL
LIN {X 0,Y 411.173,Z 353.89,A -85,B 0,C 180,E1 -10395.509,E2 -10395.509} C_VEL
LIN {X 0,Y 411.147,Z 353.896,A -85,B 0,C 180,E1 -10398.774,E2 -10398.774} C_VEL
LIN {X 0,Y 411.182,Z 353.893,A -85,B 0,C 180,E1 -10402.025,E2 -10402.025} C_VEL
LIN {X 0,Y 411.198,Z 353.887,A -85,B 0,C 180,E1 -10405.666,E2 -10405.666} C_VEL
LIN {X 0,Y 411.189,Z 353.882,A -85,B 0,C 180,E1 -10409.152,E2 -10409.152} C_VEL
LIN {X 0,Y 411.187,Z 353.879,A -85,B 0,C 180,E1 -10412.517,E2 -10412.517} C_VEL
LIN {X 0,Y 411.192,Z 353.89,A -85,B 0,C 180,E1 -10415.782,E2 -10415.782} C_VEL
LIN {X 0,Y 411.197,Z 353.881,A -85,B 0,C 180,E1 -10418.966,E2 -10418.966} C_VEL
LIN {X 0,Y 411.246,Z 353.874,A -85,B 0,C 180,E1 -10422.085,E2 -10422.085} C_VEL
LIN {X 0,Y 411.26,Z 353.877,A -85,B 0,C 180,E1 -10425.147,E2 -10425.147} C_VEL
LIN {X 0,Y 411.283,Z 353.866,A -85,B 0,C 180,E1 -10428.167,E2 -10428.167} C_VEL
LIN {X 0,Y 411.439,Z 353.857,A -85,B 0,C 180,E1 -10432.191,E2 -10432.191} C_VEL
LIN {X 0,Y 411.469,Z 353.843,A -85,B 0,C 180,E1 -10434.118,E2 -10434.118} C_VEL
LIN {X 0,Y 411.508,Z 353.849,A -85,B 0,C 180,E1 -10438.042,E2 -10438.042} C_VEL
LIN {X 0,Y 411.639,Z 353.825,A -85,B 0,C 180,E1 -10440,E2 -10440} C_VEL
LIN {X 0,Y 411.452,Z 353.848,A -85,B 0,C 180,E1 -10442.937,E2 -10442.937} C_VEL
LIN {X 0,Y 411.425,Z 353.851,A -85,B 0,C 180,E1 -10446.867,E2 -10446.867} C_VEL
LIN {X 0,Y 411.292,Z 353.875,A -85,B 0,C 180,E1 -10449.839,E2 -10449.839} C_VEL
LIN {X 0,Y 411.306,Z 353.863,A -85,B 0,C 180,E1 -10453.104,E2 -10453.104} C_VEL
LIN {X 0,Y 411.257,Z 353.881,A -85,B 0,C 180,E1 -10456.889,E2 -10456.889} C_VEL
LIN {X 0,Y 411.231,Z 353.873,A -85,B 0,C 180,E1 -10459.987,E2 -10459.987} C_VEL
LIN {X 0,Y 411.203,Z 353.888,A -85,B 0,C 180,E1 -10463.147,E2 -10463.147} C_VEL
LIN {X 0,Y 411.237,Z 353.879,A -85,B 0,C 180,E1 -10466.381,E2 -10466.381} C_VEL
LIN {X 0,Y 411.2,Z 353.877,A -85,B 0,C 180,E1 -10469.713,E2 -10469.713} C_VEL
LIN {X 0,Y 411.206,Z 353.886,A -85,B 0,C 180,E1 -10473.156,E2 -10473.156} C_VEL
LIN {X 0,Y 411.192,Z 353.89,A -85,B 0,C 180,E1 -10476.552,E2 -10476.552} C_VEL
LIN {X 0,Y 411.208,Z 353.853,A -85,B 0,C 180,E1 -10479.727,E2 -10479.727} C_VEL
LIN {X 0,Y 411.177,Z 353.892,A -85,B 0,C 180,E1 -10483.133,E2 -10483.133} C_VEL
LIN {X 0,Y 411.168,Z 353.873,A -85,B 0,C 180,E1 -10485.881,E2 -10485.881} C_VEL
LIN {X 0,Y 411.164,Z 353.889,A -85,B 0,C 180,E1 -10488.772,E2 -10488.772} C_VEL
LIN {X 0,Y 411.206,Z 353.889,A -85,B 0,C 180,E1 -10491.831,E2 -10491.831} C_VEL
LIN {X 0,Y 411.21,Z 353.887,A -85,B 0,C 180,E1 -10495.122,E2 -10495.122} C_VEL
LIN {X 0,Y 411.271,Z 354.138,A -85,B 0,C 180,E1 -10496.036,E2 -10496.036} C_VEL
LIN {X 0,Y 416.133,Z 372.145,A -85,B 0,C 180,E1 -10499.278,E2 -10499.278} C_VEL
LIN {X 0,Y 419.061,Z 383.886,A -85,B 0,C 180,E1 -10501.279,E2 -10501.279} C_VEL
LIN {X 0,Y 418.232,Z 394.372,A -85,B 0,C 180,E1 -10502.79,E2 -10502.79} C_VEL
LIN {X 0,Y 423.575,Z 426.325,A -85,B 0,C 180,E1 -10503.773,E2 -10503.773} C_VEL
LIN {X 0,Y 421.128,Z 565.209,A -85,B 0,C 180,E1 -10506.193,E2 -10506.193} C_VEL
LIN {X 0,Y 420.441,Z 581.013,A -85,B 0,C 180,E1 -10506.665,E2 -10506.665} C_VEL
LIN {X 0,Y 419.536,Z 596.337,A -85,B 0,C 180,E1 -10507.338,E2 -10507.338} C_VEL
LIN {X 0,Y 418.461,Z 610.821,A -85,B 0,C 180,E1 -10508.187,E2 -10508.187} C_VEL
LIN {X 0,Y 417.288,Z 624.014,A -85,B 0,C 180,E1 -10509.158,E2 -10509.158} C_VEL
LIN {X 0,Y 415.971,Z 637.412,A -85,B 0,C 180,E1 -10510.379,E2 -10510.379} C_VEL
LIN {X 0,Y 414.703,Z 649.94,A -85,B 0,C 180,E1 -10511.778,E2 -10511.778} C_VEL
LIN {X 0,Y 413.576,Z 660.64,A -85,B 0,C 180,E1 -10513.209,E2 -10513.209} C_VEL
LIN {X 0,Y 412.462,Z 671.364,A -85,B 0,C 180,E1 -10514.939,E2 -10514.939} C_VEL
LIN {X 0,Y 411.542,Z 680.64,A -85,B 0,C 180,E1 -10516.755,E2 -10516.755} C_VEL
LIN {X 0,Y 410.937,Z 688.584,A -85,B 0,C 180,E1 -10518.657,E2 -10518.657} C_VEL
LIN {X 0,Y 410.429,Z 695.248,A -85,B 0,C 180,E1 -10520.638,E2 -10520.638} C_VEL
LIN {X 0,Y 410.156,Z 700.451,A -85,B 0,C 180,E1 -10522.616,E2 -10522.616} C_VEL
LIN {X 0,Y 409.99,Z 703.439,A -85,B 0,C 180,E1 -10524.097,E2 -10524.097} C_VEL
LIN {X 0,Y 409.902,Z 706.365,A -85,B 0,C 180,E1 -10526.068,E2 -10526.068} C_VEL
LIN {X 0,Y 409.978,Z 708.112,A -85,B 0,C 180,E1 -10528.035,E2 -10528.035} C_VEL
LIN {X 0,Y 409.885,Z 708.709,A -85,B 0,C 180,E1 -10530,E2 -10530} C_VEL
LIN {X 0,Y 409.98,Z 708.112,A -85,B 0,C 180,E1 -10531.965,E2 -10531.965} C_VEL
LIN {X 0,Y 409.902,Z 706.365,A -85,B 0,C 180,E1 -10533.933,E2 -10533.933} C_VEL
LIN {X 0,Y 409.985,Z 703.432,A -85,B 0,C 180,E1 -10535.904,E2 -10535.904} C_VEL
LIN {X 0,Y 410.201,Z 699.245,A -85,B 0,C 180,E1 -10537.878,E2 -10537.878} C_VEL
LIN {X 0,Y 410.522,Z 693.701,A -85,B 0,C 180,E1 -10539.858,E2 -10539.858} C_VEL
LIN {X 0,Y 411.121,Z 686.641,A -85,B 0,C 180,E1 -10541.838,E2 -10541.838} C_VEL
LIN {X 0,Y 411.653,Z 679.76,A -85,B 0,C 180,E1 -10543.433,E2 -10543.433} C_VEL
LIN {X 0,Y 412.487,Z 671.334,A -85,B 0,C 180,E1 -10545.06,E2 -10545.06} C_VEL
LIN {X 0,Y 413.555,Z 660.603,A -85,B 0,C 180,E1 -10546.792,E2 -10546.792} C_VEL
LIN {X 0,Y 414.737,Z 649.773,A -85,B 0,C 180,E1 -10548.236,E2 -10548.236} C_VEL
LIN {X 0,Y 416,Z 637.346,A -85,B 0,C 180,E1 -10549.62,E2 -10549.62} C_VEL
LIN {X 0,Y 417.311,Z 623.943,A -85,B 0,C 180,E1 -10550.841,E2 -10550.841} C_VEL
LIN {X 0,Y 418.483,Z 610.739,A -85,B 0,C 180,E1 -10551.812,E2 -10551.812} C_VEL
LIN {X 0,Y 419.561,Z 596.211,A -85,B 0,C 180,E1 -10552.661,E2 -10552.661} C_VEL
LIN {X 0,Y 420.459,Z 581.236,A -85,B 0,C 180,E1 -10553.317,E2 -10553.317} C_VEL
LIN {X 0,Y 421.112,Z 566.19,A -85,B 0,C 180,E1 -10553.775,E2 -10553.775} C_VEL
LIN {X 0,Y 422.063,Z 514.371,A -85,B 0,C 180,E1 -10554.699,E2 -10554.699} C_VEL
LIN {X 0,Y 422.576,Z 493.163,A -85,B 0,C 180,E1 -10555.094,E2 -10555.094} C_VEL
LIN {X 0,Y 425.337,Z 425.612,A -85,B 0,C 180,E1 -10556.711,E2 -10556.711} C_VEL
LIN {X 0,Y 423.238,Z 410.456,A -85,B 0,C 180,E1 -10557.36,E2 -10557.36} C_VEL
LIN {X 0,Y 420.922,Z 398.598,A -85,B 0,C 180,E1 -10557.982,E2 -10557.982} C_VEL
LIN {X 0,Y 422.102,Z 390.735,A -85,B 0,C 180,E1 -10559.293,E2 -10559.293} C_VEL
LIN {X 0,Y 421.67,Z 387.281,A -85,B 0,C 180,E1 -10560.001,E2 -10560.001} C_VEL
LIN {X 0,Y 419.891,Z 379.536,A -85,B 0,C 180,E1 -10561.819,E2 -10561.819} C_VEL
LIN {X 0,Y 417.682,Z 371.753,A -85,B 0,C 180,E1 -10563.953,E2 -10563.953} C_VEL
LIN {X 0,Y 415.294,Z 364.759,A -85,B 0,C 180,E1 -10566.321,E2 -10566.321} C_VEL
LIN {X 0,Y 413.366,Z 359.638,A -85,B 0,C 180,E1 -10568.548,E2 -10568.548} C_VEL
LIN {X 0,Y 412.059,Z 356.471,A -85,B 0,C 180,E1 -10570.4,E2 -10570.4} C_VEL
LIN {X 0,Y 411.213,Z 354.003,A -85,B 0,C 180,E1 -10572.468,E2 -10572.468} C_VEL
LIN {X 0,Y 411.168,Z 353.896,A -85,B 0,C 180,E1 -10575.881,E2 -10575.881} C_VEL
LIN {X 0,Y 411.197,Z 354.054,A -85,B 0,C 180,E1 -10579.228,E2 -10579.228} C_VEL
LIN {X 0,Y 412.324,Z 356.945,A -85,B 0,C 180,E1 -10581.634,E2 -10581.634} C_VEL
LIN {X 0,Y 413.604,Z 360.189,A -85,B 0,C 180,E1 -10583.507,E2 -10583.507} C_VEL
LIN {X 0,Y 415.623,Z 366.118,A -85,B 0,C 180,E1 -10586.081,E2 -10586.081} C_VEL
LIN {X 0,Y 417.755,Z 373.333,A -85,B 0,C 180,E1 -10588.566,E2 -10588.566} C_VEL
LIN {X 0,Y 419.432,Z 380.389,A -85,B 0,C 180,E1 -10590.612,E2 -10590.612} C_VEL
LIN {X 0,Y 420.703,Z 386.919,A -85,B 0,C 180,E1 -10592.299,E2 -10592.299} C_VEL
LIN {X 0,Y 420.622,Z 389.645,A -85,B 0,C 180,E1 -10592.892,E2 -10592.892} C_VEL
LIN {X 0,Y 419.34,Z 398.753,A -85,B 0,C 180,E1 -10594.654,E2 -10594.654} C_VEL
LIN {X 0,Y 422.378,Z 411.558,A -85,B 0,C 180,E1 -10595.428,E2 -10595.428} C_VEL
LIN {X 0,Y 424.923,Z 425.258,A -85,B 0,C 180,E1 -10596.122,E2 -10596.122} C_VEL
LIN {X 0,Y 424.792,Z 430.666,A -85,B 0,C 180,E1 -10596.282,E2 -10596.282} C_VEL
LIN {X 0,Y 421.076,Z 506.35,A -85,B 0,C 180,E1 -10598.232,E2 -10598.232} C_VEL
LIN {X 0,Y 419.575,Z 544.325,A -85,B 0,C 180,E1 -10599.213,E2 -10599.213} C_VEL
LIN {X 0,Y 418.688,Z 559.707,A -85,B 0,C 180,E1 -10599.809,E2 -10599.809} C_VEL
LIN {X 0,Y 417.848,Z 573.881,A -85,B 0,C 180,E1 -10600.57,E2 -10600.57} C_VEL
LIN {X 0,Y 416.688,Z 588.253,A -85,B 0,C 180,E1 -10601.564,E2 -10601.564} C_VEL
LIN {X 0,Y 415.603,Z 600.884,A -85,B 0,C 180,E1 -10602.66,E2 -10602.66} C_VEL
LIN {X 0,Y 414.664,Z 612.434,A -85,B 0,C 180,E1 -10603.887,E2 -10603.887} C_VEL
LIN {X 0,Y 413.655,Z 622.989,A -85,B 0,C 180,E1 -10605.235,E2 -10605.235} C_VEL
LIN {X 0,Y 412.736,Z 632.582,A -85,B 0,C 180,E1 -10606.71,E2 -10606.71} C_VEL
LIN {X 0,Y 411.897,Z 641.719,A -85,B 0,C 180,E1 -10608.435,E2 -10608.435} C_VEL
LIN {X 0,Y 411.316,Z 649.081,A -85,B 0,C 180,E1 -10610.162,E2 -10610.162} C_VEL
LIN {X 0,Y 410.85,Z 654.228,A -85,B 0,C 180,E1 -10611.64,E2 -10611.64} C_VEL
LIN {X 0,Y 410.554,Z 659.232,A -85,B 0,C 180,E1 -10613.494,E2 -10613.494} C_VEL
LIN {X 0,Y 410.213,Z 662.424,A -85,B 0,C 180,E1 -10615.086,E2 -10615.086} C_VEL
LIN {X 0,Y 410.268,Z 663.891,A -85,B 0,C 180,E1 -10616.071,E2 -10616.071} C_VEL
LIN {X 0,Y 410.079,Z 665.74,A -85,B 0,C 180,E1 -10618.036,E2 -10618.036} C_VEL
LIN {X 0,Y 409.982,Z 666.158,A -85,B 0,C 180,E1 -10620,E2 -10620} C_VEL
LIN {X 0,Y 410.057,Z 665.153,A -85,B 0,C 180,E1 -10621.964,E2 -10621.964} C_VEL
LIN {X 0,Y 410.131,Z 664.118,A -85,B 0,C 180,E1 -10622.947,E2 -10622.947} C_VEL
LIN {X 0,Y 410.175,Z 660.958,A -85,B 0,C 180,E1 -10624.915,E2 -10624.915} C_VEL
LIN {X 0,Y 410.424,Z 656.266,A -85,B 0,C 180,E1 -10626.884,E2 -10626.884} C_VEL
LIN {X 0,Y 410.592,Z 651.623,A -85,B 0,C 180,E1 -10628.366,E2 -10628.366} C_VEL
LIN {X 0,Y 411.013,Z 644.895,A -85,B 0,C 180,E1 -10630.094,E2 -10630.094} C_VEL
LIN {X 0,Y 411.602,Z 636.531,A -85,B 0,C 180,E1 -10631.824,E2 -10631.824} C_VEL
LIN {X 0,Y 412.246,Z 627.357,A -85,B 0,C 180,E1 -10633.374,E2 -10633.374} C_VEL
LIN {X 0,Y 412.965,Z 617.219,A -85,B 0,C 180,E1 -10634.79,E2 -10634.79} C_VEL
LIN {X 0,Y 413.848,Z 605.405,A -85,B 0,C 180,E1 -10636.146,E2 -10636.146} C_VEL
LIN {X 0,Y 414.766,Z 592.257,A -85,B 0,C 180,E1 -10637.376,E2 -10637.376} C_VEL
LIN {X 0,Y 415.617,Z 579.227,A -85,B 0,C 180,E1 -10638.358,E2 -10638.358} C_VEL
LIN {X 0,Y 416.446,Z 565.189,A -85,B 0,C 180,E1 -10639.188,E2 -10639.188} C_VEL
LIN {X 0,Y 417.042,Z 550.801,A -85,B 0,C 180,E1 -10639.825,E2 -10639.825} C_VEL
LIN {X 0,Y 417.582,Z 535.785,A -85,B 0,C 180,E1 -10640.279,E2 -10640.279} C_VEL
LIN {X 0,Y 420.273,Z 423.931,A -85,B 0,C 180,E1 -10642.653,E2 -10642.653} C_VEL
LIN {X 0,Y 415.688,Z 397.854,A -85,B 0,C 180,E1 -10643.51,E2 -10643.51} C_VEL
LIN {X 0,Y 417.029,Z 380.992,A -85,B 0,C 180,E1 -10646.387,E2 -10646.387} C_VEL
LIN {X 0,Y 416.725,Z 377.199,A -85,B 0,C 180,E1 -10647.088,E2 -10647.088} C_VEL
LIN {X 0,Y 413.02,Z 361.504,A -85,B 0,C 180,E1 -10650.205,E2 -10650.205} C_VEL
LIN {X 0,Y 411.252,Z 354.296,A -85,B 0,C 180,E1 -10651.701,E2 -10651.701} C_VEL
LIN {X 0,Y 411.18,Z 353.895,A -85,B 0,C 180,E1 -10651.996,E2 -10651.996} C_VEL
LIN {X 0,Y 411.175,Z 353.895,A -85,B 0,C 180,E1 -10655.531,E2 -10655.531} C_VEL
LIN {X 0,Y 411.176,Z 353.891,A -85,B 0,C 180,E1 -10659.229,E2 -10659.229} C_VEL
LIN {X 0,Y 411.165,Z 353.877,A -85,B 0,C 180,E1 -10662.693,E2 -10662.693} C_VEL
LIN {X 0,Y 411.163,Z 353.888,A -85,B 0,C 180,E1 -10665.882,E2 -10665.882} C_VEL
LIN {X 0,Y 411.156,Z 353.893,A -85,B 0,C 180,E1 -10669.493,E2 -10669.493} C_VEL
LIN {X 0,Y 411.178,Z 353.895,A -85,B 0,C 180,E1 -10672.024,E2 -10672.024} C_VEL
LIN {X 0,Y 411.245,Z 354.031,A -85,B 0,C 180,E1 -10675.636,E2 -10675.636} C_VEL
LIN {X 0,Y 415.377,Z 369.211,A -85,B 0,C 180,E1 -10678.365,E2 -10678.365} C_VEL
LIN {X 0,Y 418.622,Z 382.372,A -85,B 0,C 180,E1 -10680.59,E2 -10680.59} C_VEL
LIN {X 0,Y 418.905,Z 384.266,A -85,B 0,C 180,E1 -10680.887,E2 -10680.887} C_VEL
LIN {X 0,Y 418.258,Z 396.956,A -85,B 0,C 180,E1 -10682.624,E2 -10682.624} C_VEL
LIN {X 0,Y 424.215,Z 428.017,A -85,B 0,C 180,E1 -10683.633,E2 -10683.633} C_VEL
LIN {X 0,Y 422.557,Z 524.719,A -85,B 0,C 180,E1 -10685.312,E2 -10685.312} C_VEL
LIN {X 0,Y 421.901,Z 530.564,A -85,B 0,C 180,E1 -10685.379,E2 -10685.379} C_VEL
LIN {X 0,Y 416.275,Z 549.599,A -85,B 0,C 180,E1 -10685.38,E2 -10685.38} C_VEL
LIN {X 0,Y 415.506,Z 555.45,A -85,B 0,C 180,E1 -10685.441,E2 -10685.441} C_VEL
LIN {X 0,Y 414.986,Z 571.95,A -85,B 0,C 180,E1 -10685.818,E2 -10685.818} C_VEL
LIN {X 0,Y 414.126,Z 587.4,A -85,B 0,C 180,E1 -10686.37,E2 -10686.37} C_VEL
LIN {X 0,Y 413.103,Z 602.021,A -85,B 0,C 180,E1 -10687.097,E2 -10687.097} C_VEL
LIN {X 0,Y 411.981,Z 615.418,A -85,B 0,C 180,E1 -10687.957,E2 -10687.957} C_VEL
LIN {X 0,Y 410.662,Z 629.267,A -85,B 0,C 180,E1 -10689.068,E2 -10689.068} C_VEL
LIN {X 0,Y 409.285,Z 641.871,A -85,B 0,C 180,E1 -10690.306,E2 -10690.306} C_VEL
LIN {X 0,Y 407.902,Z 654.154,A -85,B 0,C 180,E1 -10691.769,E2 -10691.769} C_VEL
LIN {X 0,Y 406.585,Z 665.663,A -85,B 0,C 180,E1 -10693.428,E2 -10693.428} C_VEL
LIN {X 0,Y 405.404,Z 675.738,A -85,B 0,C 180,E1 -10695.185,E2 -10695.185} C_VEL
LIN {X 0,Y 404.576,Z 684.109,A -85,B 0,C 180,E1 -10696.948,E2 -10696.948} C_VEL
LIN {X 0,Y 404.042,Z 690.168,A -85,B 0,C 180,E1 -10698.461,E2 -10698.461} C_VEL
LIN {X 0,Y 403.421,Z 696.793,A -85,B 0,C 180,E1 -10700.474,E2 -10700.474} C_VEL
LIN {X 0,Y 403.087,Z 701.981,A -85,B 0,C 180,E1 -10702.486,E2 -10702.486} C_VEL
LIN {X 0,Y 402.898,Z 704.965,A -85,B 0,C 180,E1 -10703.992,E2 -10703.992} C_VEL
LIN {X 0,Y 402.817,Z 707.903,A -85,B 0,C 180,E1 -10705.998,E2 -10705.998} C_VEL
LIN {X 0,Y 402.819,Z 709.665,A -85,B 0,C 180,E1 -10708,E2 -10708} C_VEL
LIN {X 0,Y 402.813,Z 710.276,A -85,B 0,C 180,E1 -10710,E2 -10710} C_VEL
LIN {X 0,Y 402.82,Z 709.707,A -85,B 0,C 180,E1 -10712,E2 -10712} C_VEL
LIN {X 0,Y 402.818,Z 708.003,A -85,B 0,C 180,E1 -10714.002,E2 -10714.002} C_VEL
LIN {X 0,Y 402.978,Z 704.734,A -85,B 0,C 180,E1 -10716.232,E2 -10716.232} C_VEL
LIN {X 0,Y 403.15,Z 701.021,A -85,B 0,C 180,E1 -10718.017,E2 -10718.017} C_VEL
LIN {X 0,Y 403.517,Z 695.564,A -85,B 0,C 180,E1 -10720.03,E2 -10720.03} C_VEL
LIN {X 0,Y 404.207,Z 688.614,A -85,B 0,C 180,E1 -10722.043,E2 -10722.043} C_VEL
LIN {X 0,Y 404.856,Z 681.045,A -85,B 0,C 180,E1 -10723.837,E2 -10723.837} C_VEL
LIN {X 0,Y 405.837,Z 672.215,A -85,B 0,C 180,E1 -10725.57,E2 -10725.57} C_VEL
LIN {X 0,Y 407.06,Z 661.385,A -85,B 0,C 180,E1 -10727.327,E2 -10727.327} C_VEL
LIN {X 0,Y 408.258,Z 650.737,A -85,B 0,C 180,E1 -10728.772,E2 -10728.772} C_VEL
LIN {X 0,Y 409.684,Z 638.072,A -85,B 0,C 180,E1 -10730.196,E2 -10730.196} C_VEL
LIN {X 0,Y 411.112,Z 624.617,A -85,B 0,C 180,E1 -10731.433,E2 -10731.433} C_VEL
LIN {X 0,Y 412.401,Z 611.468,A -85,B 0,C 180,E1 -10732.415,E2 -10732.415} C_VEL
LIN {X 0,Y 413.555,Z 596.755,A -85,B 0,C 180,E1 -10733.287,E2 -10733.287} C_VEL
LIN {X 0,Y 414.474,Z 581.787,A -85,B 0,C 180,E1 -10733.956,E2 -10733.956} C_VEL
LIN {X 0,Y 415.224,Z 566.286,A -85,B 0,C 180,E1 -10734.433,E2 -10734.433} C_VEL
LIN {X 0,Y 416.133,Z 523.787,A -85,B 0,C 180,E1 -10735.208,E2 -10735.208} C_VEL
LIN {X 0,Y 417.842,Z 428.686,A -85,B 0,C 180,E1 -10736.884,E2 -10736.884} C_VEL
LIN {X 0,Y 411.837,Z 398.041,A -85,B 0,C 180,E1 -10737.899,E2 -10737.899} C_VEL
LIN {X 0,Y 411.656,Z 396.435,A -85,B 0,C 180,E1 -10738.002,E2 -10738.002} C_VEL
LIN {X 0,Y 412.204,Z 386.915,A -85,B 0,C 180,E1 -10739.319,E2 -10739.319} C_VEL
LIN {X 0,Y 411.609,Z 382.926,A -85,B 0,C 180,E1 -10739.962,E2 -10739.962} C_VEL
LIN {X 0,Y 408.041,Z 368.496,A -85,B 0,C 180,E1 -10742.439,E2 -10742.439} C_VEL
LIN {X 0,Y 404.185,Z 354.927,A -85,B 0,C 180,E1 -10744.942,E2 -10744.942} C_VEL
LIN {X 0,Y 404.133,Z 354.764,A -85,B 0,C 180,E1 -10748.504,E2 -10748.504} C_VEL
LIN {X 0,Y 404.104,Z 354.775,A -85,B 0,C 180,E1 -10751.596,E2 -10751.596} C_VEL
LIN {X 0,Y 404.142,Z 354.765,A -85,B 0,C 180,E1 -10754.521,E2 -10754.521} C_VEL
LIN {X 0,Y 404.12,Z 354.771,A -85,B 0,C 180,E1 -10757.293,E2 -10757.293} C_VEL
LIN {X 0,Y 404.132,Z 354.769,A -85,B 0,C 180,E1 -10759.951,E2 -10759.951} C_VEL
LIN {X 0,Y 404.132,Z 354.77,A -85,B 0,C 180,E1 -10763.126,E2 -10763.126} C_VEL
LIN {X 0,Y 404.141,Z 354.769,A -85,B 0,C 180,E1 -10766.187,E2 -10766.187} C_VEL
LIN {X 0,Y 404.144,Z 354.765,A -85,B 0,C 180,E1 -10769.715,E2 -10769.715} C_VEL
LIN {X 0,Y 404.129,Z 354.757,A -85,B 0,C 180,E1 -10773.118,E2 -10773.118} C_VEL
LIN {X 0,Y 404.15,Z 354.762,A -85,B 0,C 180,E1 -10776.424,E2 -10776.424} C_VEL
LIN {X 0,Y 404.192,Z 354.764,A -85,B 0,C 180,E1 -10779.874,E2 -10779.874} C_VEL
LIN {X 0,Y 404.216,Z 354.746,A -85,B 0,C 180,E1 -10782.993,E2 -10782.993} C_VEL
LIN {X 0,Y 404.283,Z 354.749,A -85,B 0,C 180,E1 -10786.939,E2 -10786.939} C_VEL
LIN {X 0,Y 404.257,Z 354.745,A -85,B 0,C 180,E1 -10789.988,E2 -10789.988} C_VEL
LIN {X 0,Y 404.388,Z 354.737,A -85,B 0,C 180,E1 -10793.012,E2 -10793.012} C_VEL
LIN {X 0,Y 404.276,Z 354.736,A -85,B 0,C 180,E1 -10795.013,E2 -10795.013} C_VEL
LIN {X 0,Y 404.477,Z 354.726,A -85,B 0,C 180,E1 -10798.008,E2 -10798.008} C_VEL
LIN {X 0,Y 404.608,Z 354.701,A -85,B 0,C 180,E1 -10800,E2 -10800} C_VEL
LIN {X 0,Y 404.41,Z 354.725,A -85,B 0,C 180,E1 -10802.988,E2 -10802.988} C_VEL
LIN {X 0,Y 404.37,Z 354.727,A -85,B 0,C 180,E1 -10806.988,E2 -10806.988} C_VEL
LIN {X 0,Y 404.258,Z 354.75,A -85,B 0,C 180,E1 -10810.012,E2 -10810.012} C_VEL
LIN {X 0,Y 404.267,Z 354.738,A -85,B 0,C 180,E1 -10813.211,E2 -10813.211} C_VEL
LIN {X 0,Y 404.216,Z 354.76,A -85,B 0,C 180,E1 -10817.007,E2 -10817.007} C_VEL
LIN {X 0,Y 404.164,Z 354.754,A -85,B 0,C 180,E1 -10820.351,E2 -10820.351} C_VEL
LIN {X 0,Y 404.169,Z 354.759,A -85,B 0,C 180,E1 -10823.574,E2 -10823.574} C_VEL
LIN {X 0,Y 404.183,Z 354.756,A -85,B 0,C 180,E1 -10825.766,E2 -10825.766} C_VEL
LIN {X 0,Y 404.195,Z 354.76,A -85,B 0,C 180,E1 -10828,E2 -10828} C_VEL
LIN {X 0,Y 404.14,Z 354.77,A -85,B 0,C 180,E1 -10831.558,E2 -10831.558} C_VEL
LIN {X 0,Y 404.184,Z 354.756,A -85,B 0,C 180,E1 -10835.016,E2 -10835.016} C_VEL
LIN {X 0,Y 404.15,Z 354.744,A -85,B 0,C 180,E1 -10838.757,E2 -10838.757} C_VEL
LIN {X 0,Y 404.123,Z 354.747,A -85,B 0,C 180,E1 -10841.6,E2 -10841.6} C_VEL
LIN {X 0,Y 404.148,Z 354.766,A -85,B 0,C 180,E1 -10844.523,E2 -10844.523} C_VEL
LIN {X 0,Y 404.135,Z 354.744,A -85,B 0,C 180,E1 -10847.296,E2 -10847.296} C_VEL
LIN {X 0,Y 404.168,Z 354.764,A -85,B 0,C 180,E1 -10849.955,E2 -10849.955} C_VEL
LIN {X 0,Y 404.136,Z 354.77,A -85,B 0,C 180,E1 -10853.125,E2 -10853.125} C_VEL
LIN {X 0,Y 404.196,Z 354.943,A -85,B 0,C 180,E1 -10855.61,E2 -10855.61} C_VEL
LIN {X 0,Y 408.635,Z 371.414,A -85,B 0,C 180,E1 -10858.65,E2 -10858.65} C_VEL
LIN {X 0,Y 412.111,Z 385.046,A -85,B 0,C 180,E1 -10861.027,E2 -10861.027} C_VEL
LIN {X 0,Y 412.154,Z 387.958,A -85,B 0,C 180,E1 -10861.481,E2 -10861.481} C_VEL
LIN {X 0,Y 411.623,Z 393.739,A -85,B 0,C 180,E1 -10862.301,E2 -10862.301} C_VEL
LIN {X 0,Y 417.183,Z 426.733,A -85,B 0,C 180,E1 -10863.345,E2 -10863.345} C_VEL
LIN {X 0,Y 415.003,Z 549.008,A -85,B 0,C 180,E1 -10865.487,E2 -10865.487} C_VEL
LIN {X 0,Y 414.513,Z 568.777,A -85,B 0,C 180,E1 -10865.889,E2 -10865.889} C_VEL
LIN {X 0,Y 413.809,Z 583.746,A -85,B 0,C 180,E1 -10866.385,E2 -10866.385} C_VEL
LIN {X 0,Y 412.921,Z 597.505,A -85,B 0,C 180,E1 -10867.021,E2 -10867.021} C_VEL
LIN {X 0,Y 411.876,Z 610.861,A -85,B 0,C 180,E1 -10867.819,E2 -10867.819} C_VEL
LIN {X 0,Y 410.618,Z 624.047,A -85,B 0,C 180,E1 -10868.804,E2 -10868.804} C_VEL
LIN {X 0,Y 409.274,Z 637.44,A -85,B 0,C 180,E1 -10870.045,E2 -10870.045} C_VEL
LIN {X 0,Y 408.082,Z 648.649,A -85,B 0,C 180,E1 -10871.3,E2 -10871.3} C_VEL
LIN {X 0,Y 406.731,Z 660.662,A -85,B 0,C 180,E1 -10872.918,E2 -10872.918} C_VEL
LIN {X 0,Y 405.557,Z 671.385,A -85,B 0,C 180,E1 -10874.676,E2 -10874.676} C_VEL
LIN {X 0,Y 404.626,Z 680.309,A -85,B 0,C 180,E1 -10876.444,E2 -10876.444} C_VEL
LIN {X 0,Y 403.943,Z 688.601,A -85,B 0,C 180,E1 -10878.458,E2 -10878.458} C_VEL
LIN {X 0,Y 403.378,Z 695.264,A -85,B 0,C 180,E1 -10880.473,E2 -10880.473} C_VEL
LIN {X 0,Y 403.083,Z 700.467,A -85,B 0,C 180,E1 -10882.486,E2 -10882.486} C_VEL
LIN {X 0,Y 402.916,Z 703.453,A -85,B 0,C 180,E1 -10883.993,E2 -10883.993} C_VEL
LIN {X 0,Y 402.822,Z 706.38,A -85,B 0,C 180,E1 -10885.998,E2 -10885.998} C_VEL
LIN {X 0,Y 402.874,Z 708.126,A -85,B 0,C 180,E1 -10888.001,E2 -10888.001} C_VEL
LIN {X 0,Y 402.812,Z 708.722,A -85,B 0,C 180,E1 -10890,E2 -10890} C_VEL
LIN {X 0,Y 402.876,Z 708.126,A -85,B 0,C 180,E1 -10892,E2 -10892} C_VEL
LIN {X 0,Y 402.822,Z 706.379,A -85,B 0,C 180,E1 -10894.002,E2 -10894.002} C_VEL
LIN {X 0,Y 402.939,Z 703.135,A -85,B 0,C 180,E1 -10896.182,E2 -10896.182} C_VEL
LIN {X 0,Y 403.142,Z 699.259,A -85,B 0,C 180,E1 -10898.017,E2 -10898.017} C_VEL
LIN {X 0,Y 403.482,Z 693.715,A -85,B 0,C 180,E1 -10900.031,E2 -10900.031} C_VEL
LIN {X 0,Y 404.13,Z 686.656,A -85,B 0,C 180,E1 -10902.045,E2 -10902.045} C_VEL
LIN {X 0,Y 404.788,Z 678.967,A -85,B 0,C 180,E1 -10903.835,E2 -10903.835} C_VEL
LIN {X 0,Y 405.713,Z 669.937,A -85,B 0,C 180,E1 -10905.575,E2 -10905.575} C_VEL
LIN {X 0,Y 406.712,Z 660.621,A -85,B 0,C 180,E1 -10907.083,E2 -10907.083} C_VEL
LIN {X 0,Y 408.103,Z 648.51,A -85,B 0,C 180,E1 -10908.709,E2 -10908.709} C_VEL
LIN {X 0,Y 409.397,Z 636.135,A -85,B 0,C 180,E1 -10910.08,E2 -10910.08} C_VEL
LIN {X 0,Y 410.803,Z 622.419,A -85,B 0,C 180,E1 -10911.318,E2 -10911.318} C_VEL
LIN {X 0,Y 412.061,Z 608.885,A -85,B 0,C 180,E1 -10912.302,E2 -10912.302} C_VEL
LIN {X 0,Y 413.109,Z 595.258,A -85,B 0,C 180,E1 -10913.09,E2 -10913.09} C_VEL
LIN {X 0,Y 414.007,Z 580.148,A -85,B 0,C 180,E1 -10913.748,E2 -10913.748} C_VEL
LIN {X 0,Y 414.703,Z 564.982,A -85,B 0,C 180,E1 -10914.199,E2 -10914.199} C_VEL
LIN {X 0,Y 415.844,Z 507.163,A -85,B 0,C 180,E1 -10915.261,E2 -10915.261} C_VEL
LIN {X 0,Y 419.418,Z 430.053,A -85,B 0,C 180,E1 -10917.137,E2 -10917.137} C_VEL
LIN {X 0,Y 419.344,Z 425.552,A -85,B 0,C 180,E1 -10917.28,E2 -10917.28} C_VEL
LIN {X 0,Y 417.324,Z 411.261,A -85,B 0,C 180,E1 -10917.928,E2 -10917.928} C_VEL
LIN {X 0,Y 414.877,Z 398.588,A -85,B 0,C 180,E1 -10918.644,E2 -10918.644} C_VEL
LIN {X 0,Y 415.764,Z 392.745,A -85,B 0,C 180,E1 -10919.655,E2 -10919.655} C_VEL
LIN {X 0,Y 414.252,Z 384.807,A -85,B 0,C 180,E1 -10921.493,E2 -10921.493} C_VEL
LIN {X 0,Y 412.09,Z 376.859,A -85,B 0,C 180,E1 -10923.66,E2 -10923.66} C_VEL
LIN {X 0,Y 410.179,Z 370.9,A -85,B 0,C 180,E1 -10925.631,E2 -10925.631} C_VEL
LIN {X 0,Y 408.418,Z 365.853,A -85,B 0,C 180,E1 -10927.668,E2 -10927.668} C_VEL
LIN {X 0,Y 406.97,Z 361.919,A -85,B 0,C 180,E1 -10929.714,E2 -10929.714} C_VEL
LIN {X 0,Y 405.632,Z 358.376,A -85,B 0,C 180,E1 -10932.51,E2 -10932.51} C_VEL
LIN {X 0,Y 404.942,Z 357.259,A -85,B 0,C 180,E1 -10934.637,E2 -10934.637} C_VEL
LIN {X 0,Y 404.892,Z 357.204,A -85,B 0,C 180,E1 -10936.805,E2 -10936.805} C_VEL
LIN {X 0,Y 405.451,Z 358.095,A -85,B 0,C 180,E1 -10938.801,E2 -10938.801} C_VEL
LIN {X 0,Y 406.592,Z 361.101,A -85,B 0,C 180,E1 -10941.518,E2 -10941.518} C_VEL
LIN {X 0,Y 408.165,Z 365.484,A -85,B 0,C 180,E1 -10944.025,E2 -10944.025} C_VEL
LIN {X 0,Y 409.946,Z 370.87,A -85,B 0,C 180,E1 -10946.35,E2 -10946.35} C_VEL
LIN {X 0,Y 412.027,Z 378.486,A -85,B 0,C 180,E1 -10948.968,E2 -10948.968} C_VEL
LIN {X 0,Y 413.844,Z 386.76,A -85,B 0,C 180,E1 -10951.334,E2 -10951.334} C_VEL
LIN {X 0,Y 414.338,Z 391.409,A -85,B 0,C 180,E1 -10952.494,E2 -10952.494} C_VEL
LIN {X 0,Y 413.231,Z 398.839,A -85,B 0,C 180,E1 -10953.961,E2 -10953.961} C_VEL
LIN {X 0,Y 416.433,Z 412.485,A -85,B 0,C 180,E1 -10954.843,E2 -10954.843} C_VEL
LIN {X 0,Y 419.046,Z 426.525,A -85,B 0,C 180,E1 -10955.597,E2 -10955.597} C_VEL
LIN {X 0,Y 418.818,Z 433.159,A -85,B 0,C 180,E1 -10955.796,E2 -10955.796} C_VEL
LIN {X 0,Y 414.8,Z 507.944,A -85,B 0,C 180,E1 -10957.788,E2 -10957.788} C_VEL
LIN {X 0,Y 413.233,Z 544.899,A -85,B 0,C 180,E1 -10958.781,E2 -10958.781} C_VEL
LIN {X 0,Y 412.275,Z 560.705,A -85,B 0,C 180,E1 -10959.416,E2 -10959.416} C_VEL
LIN {X 0,Y 411.273,Z 575.545,A -85,B 0,C 180,E1 -10960.247,E2 -10960.247} C_VEL
LIN {X 0,Y 410.077,Z 589.591,A -85,B 0,C 180,E1 -10961.256,E2 -10961.256} C_VEL
LIN {X 0,Y 408.931,Z 602.017,A -85,B 0,C 180,E1 -10962.368,E2 -10962.368} C_VEL
LIN {X 0,Y 407.914,Z 613.415,A -85,B 0,C 180,E1 -10963.613,E2 -10963.613} C_VEL
LIN {X 0,Y 406.855,Z 623.859,A -85,B 0,C 180,E1 -10964.983,E2 -10964.983} C_VEL
LIN {X 0,Y 405.864,Z 633.359,A -85,B 0,C 180,E1 -10966.481,E2 -10966.481} C_VEL
LIN {X 0,Y 404.969,Z 642.396,A -85,B 0,C 180,E1 -10968.234,E2 -10968.234} C_VEL
LIN {X 0,Y 404.323,Z 649.7,A -85,B 0,C 180,E1 -10969.99,E2 -10969.99} C_VEL
LIN {X 0,Y 403.851,Z 654.796,A -85,B 0,C 180,E1 -10971.494,E2 -10971.494} C_VEL
LIN {X 0,Y 403.519,Z 659.123,A -85,B 0,C 180,E1 -10973.101,E2 -10973.101} C_VEL
LIN {X 0,Y 403.155,Z 662.916,A -85,B 0,C 180,E1 -10975,E2 -10975} C_VEL
LIN {X 0,Y 403.196,Z 664.349,A -85,B 0,C 180,E1 -10976.002,E2 -10976.002} C_VEL
LIN {X 0,Y 403.01,Z 666.14,A -85,B 0,C 180,E1 -10978.001,E2 -10978.001} C_VEL
LIN {X 0,Y 402.904,Z 666.505,A -85,B 0,C 180,E1 -10980,E2 -10980} C_VEL
LIN {X 0,Y 402.988,Z 665.442,A -85,B 0,C 180,E1 -10981.999,E2 -10981.999} C_VEL
LIN {X 0,Y 403.048,Z 664.376,A -85,B 0,C 180,E1 -10982.999,E2 -10982.999} C_VEL
LIN {X 0,Y 403.118,Z 661.149,A -85,B 0,C 180,E1 -10985.001,E2 -10985.001} C_VEL
LIN {X 0,Y 403.356,Z 656.381,A -85,B 0,C 180,E1 -10987.006,E2 -10987.006} C_VEL
LIN {X 0,Y 403.537,Z 651.662,A -85,B 0,C 180,E1 -10988.513,E2 -10988.513} C_VEL
LIN {X 0,Y 404.001,Z 644.842,A -85,B 0,C 180,E1 -10990.271,E2 -10990.271} C_VEL
LIN {X 0,Y 404.611,Z 636.373,A -85,B 0,C 180,E1 -10992.031,E2 -10992.031} C_VEL
LIN {X 0,Y 405.309,Z 626.747,A -85,B 0,C 180,E1 -10993.654,E2 -10993.654} C_VEL
LIN {X 0,Y 406.109,Z 615.756,A -85,B 0,C 180,E1 -10995.174,E2 -10995.174} C_VEL
LIN {X 0,Y 407.029,Z 603.586,A -85,B 0,C 180,E1 -10996.553,E2 -10996.553} C_VEL
LIN {X 0,Y 407.946,Z 591.459,A -85,B 0,C 180,E1 -10997.676,E2 -10997.676} C_VEL
LIN {X 0,Y 408.832,Z 578.18,A -85,B 0,C 180,E1 -10998.673,E2 -10998.673} C_VEL
LIN {X 0,Y 409.617,Z 564.143,A -85,B 0,C 180,E1 -10999.494,E2 -10999.494} C_VEL
LIN {X 0,Y 410.285,Z 549.529,A -85,B 0,C 180,E1 -11000.133,E2 -11000.133} C_VEL
LIN {X 0,Y 410.81,Z 533.893,A -85,B 0,C 180,E1 -11000.596,E2 -11000.596} C_VEL
LIN {X 0,Y 413.668,Z 425.428,A -85,B 0,C 180,E1 -11002.953,E2 -11002.953} C_VEL
LIN {X 0,Y 408.881,Z 397.842,A -85,B 0,C 180,E1 -11003.876,E2 -11003.876} C_VEL
LIN {X 0,Y 410.216,Z 381.074,A -85,B 0,C 180,E1 -11006.791,E2 -11006.791} C_VEL
LIN {X 0,Y 407.588,Z 369.184,A -85,B 0,C 180,E1 -11009.151,E2 -11009.151} C_VEL
LIN {X 0,Y 404.206,Z 355.158,A -85,B 0,C 180,E1 -11012.062,E2 -11012.062} C_VEL
LIN {X 0,Y 404.138,Z 354.815,A -85,B 0,C 180,E1 -11012.206,E2 -11012.206} C_VEL
LIN {X 0,Y 404.143,Z 354.769,A -85,B 0,C 180,E1 -11015.182,E2 -11015.182} C_VEL
LIN {X 0,Y 404.132,Z 354.77,A -85,B 0,C 180,E1 -11018.76,E2 -11018.76} C_VEL
LIN {X 0,Y 404.105,Z 354.764,A -85,B 0,C 180,E1 -11021.597,E2 -11021.597} C_VEL
LIN {X 0,Y 404.143,Z 354.771,A -85,B 0,C 180,E1 -11024.521,E2 -11024.521} C_VEL
LIN {X 0,Y 404.119,Z 354.757,A -85,B 0,C 180,E1 -11027.293,E2 -11027.293} C_VEL
LIN {X 0,Y 404.133,Z 354.762,A -85,B 0,C 180,E1 -11029.951,E2 -11029.951} C_VEL
LIN {X 0,Y 404.13,Z 354.762,A -85,B 0,C 180,E1 -11033.126,E2 -11033.126} C_VEL
LIN {X 0,Y 404.201,Z 354.956,A -85,B 0,C 180,E1 -11035.175,E2 -11035.175} C_VEL
LIN {X 0,Y 408.382,Z 369.889,A -85,B 0,C 180,E1 -11037.906,E2 -11037.906} C_VEL
LIN {X 0,Y 412.019,Z 384.775,A -85,B 0,C 180,E1 -11040.451,E2 -11040.451} C_VEL
LIN {X 0,Y 412.102,Z 388.319,A -85,B 0,C 180,E1 -11040.979,E2 -11040.979} C_VEL
LIN {X 0,Y 411.698,Z 397.169,A -85,B 0,C 180,E1 -11042.167,E2 -11042.167} C_VEL
LIN {X 0,Y 417.849,Z 429.097,A -85,B 0,C 180,E1 -11043.222,E2 -11043.222} C_VEL
LIN {X 0,Y 415.542,Z 554.222,A -85,B 0,C 180,E1 -11045.421,E2 -11045.421} C_VEL
LIN {X 0,Y 415.506,Z 555.45,A -85,B 0,C 180,E1 -11045.441,E2 -11045.441} C_VEL
LIN {X 0,Y 414.693,Z 561.302,A -85,B 0,C 180,E1 -11045.51,E2 -11045.51} C_VEL
LIN {X 0,Y 411.652,Z 570.768,A -85,B 0,C 180,E1 -11045.572,E2 -11045.572} C_VEL
LIN {X 0,Y 408.585,Z 580.14,A -85,B 0,C 180,E1 -11045.71,E2 -11045.71} C_VEL
LIN {X 0,Y 407.742,Z 585.778,A -85,B 0,C 180,E1 -11045.903,E2 -11045.903} C_VEL
LIN {X 0,Y 406.652,Z 600.899,A -85,B 0,C 180,E1 -11046.645,E2 -11046.645} C_VEL
LIN {X 0,Y 405.384,Z 615.39,A -85,B 0,C 180,E1 -11047.579,E2 -11047.579} C_VEL
LIN {X 0,Y 404.004,Z 629.243,A -85,B 0,C 180,E1 -11048.707,E2 -11048.707} C_VEL
LIN {X 0,Y 402.585,Z 641.851,A -85,B 0,C 180,E1 -11049.965,E2 -11049.965} C_VEL
LIN {X 0,Y 401.193,Z 653.556,A -85,B 0,C 180,E1 -11051.373,E2 -11051.373} C_VEL
LIN {X 0,Y 399.908,Z 664.044,A -85,B 0,C 180,E1 -11052.88,E2 -11052.88} C_VEL
LIN {X 0,Y 398.647,Z 674.388,A -85,B 0,C 180,E1 -11054.666,E2 -11054.666} C_VEL
LIN {X 0,Y 397.707,Z 682.706,A -85,B 0,C 180,E1 -11056.391,E2 -11056.391} C_VEL
LIN {X 0,Y 397.039,Z 690.154,A -85,B 0,C 180,E1 -11058.255,E2 -11058.255} C_VEL
LIN {X 0,Y 396.365,Z 696.779,A -85,B 0,C 180,E1 -11060.302,E2 -11060.302} C_VEL
LIN {X 0,Y 396.02,Z 701.967,A -85,B 0,C 180,E1 -11062.351,E2 -11062.351} C_VEL
LIN {X 0,Y 395.821,Z 704.951,A -85,B 0,C 180,E1 -11063.884,E2 -11063.884} C_VEL
LIN {X 0,Y 395.74,Z 707.889,A -85,B 0,C 180,E1 -11065.926,E2 -11065.926} C_VEL
LIN {X 0,Y 395.716,Z 709.651,A -85,B 0,C 180,E1 -11067.964,E2 -11067.964} C_VEL
LIN {X 0,Y 395.725,Z 710.262,A -85,B 0,C 180,E1 -11070,E2 -11070} C_VEL
LIN {X 0,Y 395.716,Z 709.693,A -85,B 0,C 180,E1 -11072.035,E2 -11072.035} C_VEL
LIN {X 0,Y 395.742,Z 707.989,A -85,B 0,C 180,E1 -11074.073,E2 -11074.073} C_VEL
LIN {X 0,Y 395.898,Z 704.937,A -85,B 0,C 180,E1 -11076.218,E2 -11076.218} C_VEL
LIN {X 0,Y 396.082,Z 701.005,A -85,B 0,C 180,E1 -11078.161,E2 -11078.161} C_VEL
LIN {X 0,Y 396.459,Z 695.547,A -85,B 0,C 180,E1 -11080.211,E2 -11080.211} C_VEL
LIN {X 0,Y 397.205,Z 688.596,A -85,B 0,C 180,E1 -11082.258,E2 -11082.258} C_VEL
LIN {X 0,Y 397.898,Z 681.189,A -85,B 0,C 180,E1 -11084.048,E2 -11084.048} C_VEL
LIN {X 0,Y 398.929,Z 672.193,A -85,B 0,C 180,E1 -11085.847,E2 -11085.847} C_VEL
LIN {X 0,Y 400.255,Z 661.361,A -85,B 0,C 180,E1 -11087.631,E2 -11087.631} C_VEL
LIN {X 0,Y 401.63,Z 649.778,A -85,B 0,C 180,E1 -11089.212,E2 -11089.212} C_VEL
LIN {X 0,Y 403,Z 638.041,A -85,B 0,C 180,E1 -11090.546,E2 -11090.546} C_VEL
